    |   movel(pose_trans(ref_frame,p[0.110397, 0.057635, -0.000125, -0.013708, 3.141563, -0.000000]),accel_mss,speed_ms,0,0.001)
    |   movel(pose_trans(ref_frame,p[0.110185, 0.057584, -0.000125, -0.013708, 3.141563, -0.000000]),accel_mss,speed_ms,0,0.001)
    |   movel(pose_trans(ref_frame,p[0.106841, 0.057587, -0.000125, -0.013708, 3.141563, -0.000000]),accel_mss,speed_ms,0,0.001)
    |   movel(pose_trans(ref_frame,p[0.103498, 0.057593, -0.000125, -0.013708, 3.141563, -0.000000]),accel_mss,speed_ms,0,0.001)
    |   movel(pose_trans(ref_frame,p[0.100318, 0.057604, -0.000125, -0.013708, 3.141563, -0.000000]),accel_mss,speed_ms,0,0.001)
    |   movel(pose_trans(ref_frame,p[0.097137, 0.057625, -0.000125, -0.013708, 3.141563, 0.000000]),accel_mss,speed_ms,0,0.001)
    |   movel(pose_trans(ref_frame,p[0.096513, 0.057673, -0.000125, -0.013708, 3.141563, 0.000000]),accel_mss,speed_ms,0,0.001)
    |   movel(pose_trans(ref_frame,p[0.095902, 0.057808, -0.000125, -0.013708, 3.141563, 0.000000]),accel_mss,speed_ms,0,0.001)
    |   movel(pose_trans(ref_frame,p[0.094724, 0.058284, -0.000125, -0.013708, 3.141563, -0.000000]),accel_mss,speed_ms,0,0.001)
    |   movel(pose_trans(ref_frame,p[0.093662, 0.058981, -0.000125, -0.013708, 3.141563, 0.000000]),accel_mss,speed_ms,0,0.001)
    |   movel(pose_trans(ref_frame,p[0.092768, 0.059865, -0.000125, -0.013708, 3.141563, -0.000000]),accel_mss,speed_ms,0,0.001)
    |   movel(pose_trans(ref_frame,p[0.092068, 0.060911, -0.000125, -0.013708, 3.141563, -0.000000]),accel_mss,speed_ms,0,0.001)
    |   movel(pose_trans(ref_frame,p[0.091599, 0.062063, -0.000125, -0.013708, 3.141563, -0.000000]),accel_mss,speed_ms,0,0.001)
    |   movel(pose_trans(ref_frame,p[0.091375, 0.063287, -0.000125, -0.013708, 3.141563, 0.000000]),accel_mss,speed_ms,0,0.001)
    |   movel(pose_trans(ref_frame,p[0.091405, 0.064523, -0.000125, -0.013708, 3.141563, 0.000000]),accel_mss,speed_ms,0,0.001)
    |   movel(pose_trans(ref_frame,p[0.091691, 0.065727, -0.000125, -0.013708, 3.141563, 0.000000]),accel_mss,speed_ms,0,0.001)
    |   movel(pose_trans(ref_frame,p[0.091870, 0.066190, -0.000125, -0.013708, 3.141563, -0.000000]),accel_mss,speed_ms,0,0.001)
    |   movel(pose_trans(ref_frame,p[0.092079, 0.066640, -0.000125, -0.013708, 3.141563, -0.000000]),accel_mss,speed_ms,0,0.001)
    |   movel(pose_trans(ref_frame,p[0.092300, 0.067034, -0.000125, -0.013708, 3.141563, -0.000000]),accel_mss,speed_ms,0,0.001)
    |   movel(pose_trans(ref_frame,p[0.092554, 0.067407, -0.000125, -0.013708, 3.141563, -0.000000]),accel_mss,speed_ms,0,0.001)
    |   movel(pose_trans(ref_frame,p[0.092839, 0.067757, -0.000125, -0.013708, 3.141563, -0.000000]),accel_mss,speed_ms,0,0.001)
    |   movel(pose_trans(ref_frame,p[0.093154, 0.068082, -0.000125, -0.013708, 3.141563, -0.000000]),accel_mss,speed_ms,0,0.001)
    |   movel(pose_trans(ref_frame,p[0.093526, 0.068412, -0.000125, -0.013708, 3.141563, -0.000000]),accel_mss,speed_ms,0,0.001)
    |   movel(pose_trans(ref_frame,p[0.093919, 0.068718, -0.000125, -0.013708, 3.141563, -0.000000]),accel_mss,speed_ms,0,0) # end trace
    |   speed_ms    = 1.000
    |   movel(pose_trans(ref_frame,p[0.093921, 0.068718, 0.005000, -0.013708, 3.141563, -0.000000]),accel_mss,speed_ms,0,0.001)
    |   movel(pose_trans(ref_frame,p[0.109466, 0.038489, 0.005000, -0.013708, 3.141563, -0.000000]),accel_mss,speed_ms,0,0) # end trace
    |   speed_ms    = 0.002
    |   movel(pose_trans(ref_frame,p[0.109466, 0.038489, -0.000125, -0.013708, 3.141563, 0.000000]),accel_mss,speed_ms,0,0) # end trace
    |   speed_ms    = 0.007
    |   movel(pose_trans(ref_frame,p[0.109569, 0.038507, -0.000125, -0.013708, 3.141563, -0.000000]),accel_mss,speed_ms,0,0.001)
    |   movel(pose_trans(ref_frame,p[0.109673, 0.038505, -0.000125, -0.013708, 3.141563, 0.000000]),accel_mss,speed_ms,0,0.001)
    |   movel(pose_trans(ref_frame,p[0.109805, 0.038481, -0.000125, -0.013708, 3.141563, -0.000000]),accel_mss,speed_ms,0,0.001)
    |   movel(pose_trans(ref_frame,p[0.109934, 0.038445, -0.000125, -0.013708, 3.141563, -0.000000]),accel_mss,speed_ms,0,0.001)
    |   movel(pose_trans(ref_frame,p[0.110111, 0.038380, -0.000125, -0.013708, 3.141563, -0.000000]),accel_mss,speed_ms,0,0.001)
    |   movel(pose_trans(ref_frame,p[0.110284, 0.038303, -0.000125, -0.013708, 3.141563, -0.000000]),accel_mss,speed_ms,0,0.001)
    |   movel(pose_trans(ref_frame,p[0.110541, 0.038176, -0.000125, -0.013708, 3.141563, -0.000000]),accel_mss,speed_ms,0,0.001)
    |   movel(pose_trans(ref_frame,p[0.110795, 0.038045, -0.000125, -0.013708, 3.141563, -0.000000]),accel_mss,speed_ms,0,0.001)
    |   movel(pose_trans(ref_frame,p[0.111492, 0.037703, -0.000125, -0.013708, 3.141563, -0.000000]),accel_mss,speed_ms,0,0.001)
    |   movel(pose_trans(ref_frame,p[0.112210, 0.037408, -0.000125, -0.013708, 3.141563, 0.000000]),accel_mss,speed_ms,0,0.001)
    |   movel(pose_trans(ref_frame,p[0.112732, 0.037267, -0.000125, -0.013708, 3.141563, -0.000000]),accel_mss,speed_ms,0,0.001)
    |   movel(pose_trans(ref_frame,p[0.113270, 0.037223, -0.000125, -0.013708, 3.141563, 0.000000]),accel_mss,speed_ms,0,0.001)
    |   movel(pose_trans(ref_frame,p[0.113818, 0.037279, -0.000125, -0.013708, 3.141563, -0.000000]),accel_mss,speed_ms,0,0.001)
    |   movel(pose_trans(ref_frame,p[0.114348, 0.037432, -0.000125, -0.013708, 3.141563, -0.000000]),accel_mss,speed_ms,0,0.001)
    |   movel(pose_trans(ref_frame,p[0.115100, 0.037748, -0.000125, -0.013708, 3.141563, 0.000000]),accel_mss,speed_ms,0,0.001)
    |   movel(pose_trans(ref_frame,p[0.115833, 0.038108, -0.000125, -0.013708, 3.141563, -0.000000]),accel_mss,speed_ms,0,0.001)
    |   movel(pose_trans(ref_frame,p[0.116136, 0.038265, -0.000125, -0.013708, 3.141563, 0.000000]),accel_mss,speed_ms,0,0.001)
    |   movel(pose_trans(ref_frame,p[0.116441, 0.038419, -0.000125, -0.013708, 3.141563, -0.000000]),accel_mss,speed_ms,0,0.001)
    |   movel(pose_trans(ref_frame,p[0.116571, 0.038472, -0.000125, -0.013708, 3.141563, -0.000000]),accel_mss,speed_ms,0,0.001)
    |   movel(pose_trans(ref_frame,p[0.116708, 0.038508, -0.000125, -0.013708, 3.141563, 0.000000]),accel_mss,speed_ms,0,0.001)
    |   movel(pose_trans(ref_frame,p[0.116813, 0.038515, -0.000125, -0.013708, 3.141563, -0.000000]),accel_mss,speed_ms,0,0.001)
    |   movel(pose_trans(ref_frame,p[0.116916, 0.038493, -0.000125, -0.013708, 3.141563, 0.000000]),accel_mss,speed_ms,0,0.001)
    |   movel(pose_trans(ref_frame,p[0.117051, 0.038438, -0.000125, -0.013708, 3.141563, 0.000000]),accel_mss,speed_ms,0,0.001)
    |   movel(pose_trans(ref_frame,p[0.117180, 0.038369, -0.000125, -0.013708, 3.141563, 0.000000]),accel_mss,speed_ms,0,0.001)
    |   movel(pose_trans(ref_frame,p[0.117339, 0.038252, -0.000125, -0.013708, 3.141563, -0.000000]),accel_mss,speed_ms,0,0.001)
    |   movel(pose_trans(ref_frame,p[0.117471, 0.038106, -0.000125, -0.013708, 3.141563, -0.000000]),accel_mss,speed_ms,0,0.001)
    |   movel(pose_trans(ref_frame,p[0.117545, 0.037961, -0.000125, -0.013708, 3.141563, -0.000000]),accel_mss,speed_ms,0,0.001)
    |   movel(pose_trans(ref_frame,p[0.117566, 0.037799, -0.000125, -0.013708, 3.141563, 0.000000]),accel_mss,speed_ms,0,0.001)
    |   movel(pose_trans(ref_frame,p[0.117537, 0.037580, -0.000125, -0.013708, 3.141563, 0.000000]),accel_mss,speed_ms,0,0.001)
    |   movel(pose_trans(ref_frame,p[0.117466, 0.037370, -0.000125, -0.013708, 3.141563, 0.000000]),accel_mss,speed_ms,0,0.001)
    |   movel(pose_trans(ref_frame,p[0.117297, 0.037011, -0.000125, -0.013708, 3.141563, -0.000000]),accel_mss,speed_ms,0,0.001)
    |   movel(pose_trans(ref_frame,p[0.117115, 0.036659, -0.000125, -0.013708, 3.141563, -0.000000]),accel_mss,speed_ms,0,0.001)
    |   movel(pose_trans(ref_frame,p[0.116779, 0.035981, -0.000125, -0.013708, 3.141563, -0.000000]),accel_mss,speed_ms,0,0.001)
    |   movel(pose_trans(ref_frame,p[0.116493, 0.035281, -0.000125, -0.013708, 3.141563, -0.000000]),accel_mss,speed_ms,0,0.001)
    |   movel(pose_trans(ref_frame,p[0.116347, 0.034741, -0.000125, -0.013708, 3.141563, -0.000000]),accel_mss,speed_ms,0,0.001)
    |   movel(pose_trans(ref_frame,p[0.116298, 0.034183, -0.000125, -0.013708, 3.141563, -0.000000]),accel_mss,speed_ms,0,0.001)
    |   movel(pose_trans(ref_frame,p[0.116347, 0.033625, -0.000125, -0.013708, 3.141563, -0.000000]),accel_mss,speed_ms,0,0.001)
    |   movel(pose_trans(ref_frame,p[0.116492, 0.033084, -0.000125, -0.013708, 3.141563, -0.000000]),accel_mss,speed_ms,0,0.001)
    |   movel(pose_trans(ref_frame,p[0.116778, 0.032382, -0.000125, -0.013708, 3.141563, 0.000000]),accel_mss,speed_ms,0,0.001)
    |   movel(pose_trans(ref_frame,p[0.117114, 0.031703, -0.000125, -0.013708, 3.141563, 0.000000]),accel_mss,speed_ms,0,0.001)
    |   movel(pose_trans(ref_frame,p[0.117282, 0.031378, -0.000125, -0.013708, 3.141563, -0.000000]),accel_mss,speed_ms,0,0.001)
    |   movel(pose_trans(ref_frame,p[0.117440, 0.031048, -0.000125, -0.013708, 3.141563, -0.000000]),accel_mss,speed_ms,0,0.001)
    |   movel(pose_trans(ref_frame,p[0.117514, 0.030847, -0.000125, -0.013708, 3.141563, -0.000000]),accel_mss,speed_ms,0,0.001)
    |   movel(pose_trans(ref_frame,p[0.117557, 0.030638, -0.000125, -0.013708, 3.141563, -0.000000]),accel_mss,speed_ms,0,0.001)
    |   movel(pose_trans(ref_frame,p[0.117557, 0.030481, -0.000125, -0.013708, 3.141563, 0.000000]),accel_mss,speed_ms,0,0.001)
    |   movel(pose_trans(ref_frame,p[0.117517, 0.030329, -0.000125, -0.013708, 3.141563, -0.000000]),accel_mss,speed_ms,0,0.001)
    |   movel(pose_trans(ref_frame,p[0.117437, 0.030178, -0.000125, -0.013708, 3.141563, -0.000000]),accel_mss,speed_ms,0,0.001)
    |   movel(pose_trans(ref_frame,p[0.117328, 0.030045, -0.000125, -0.013708, 3.141563, -0.000000]),accel_mss,speed_ms,0,0.001)
    |   movel(pose_trans(ref_frame,p[0.117199, 0.029939, -0.000125, -0.013708, 3.141563, -0.000000]),accel_mss,speed_ms,0,0.001)
    |   movel(pose_trans(ref_frame,p[0.117052, 0.029858, -0.000125, -0.013708, 3.141563, -0.000000]),accel_mss,speed_ms,0,0.001)
    |   movel(pose_trans(ref_frame,p[0.116906, 0.029817, -0.000125, -0.013708, 3.141563, -0.000000]),accel_mss,speed_ms,0,0.001)
    |   movel(pose_trans(ref_frame,p[0.116754, 0.029814, -0.000125, -0.013708, 3.141563, -0.000000]),accel_mss,speed_ms,0,0.001)
    |   movel(pose_trans(ref_frame,p[0.116560, 0.029851, -0.000125, -0.013708, 3.141563, -0.000000]),accel_mss,speed_ms,0,0.001)
    |   movel(pose_trans(ref_frame,p[0.116375, 0.029919, -0.000125, -0.013708, 3.141563, -0.000000]),accel_mss,speed_ms,0,0.001)
    |   movel(pose_trans(ref_frame,p[0.116090, 0.030059, -0.000125, -0.013708, 3.141563, -0.000000]),accel_mss,speed_ms,0,0.001)
    |   movel(pose_trans(ref_frame,p[0.115811, 0.030210, -0.000125, -0.013708, 3.141563, -0.000000]),accel_mss,speed_ms,0,0.001)
    |   movel(pose_trans(ref_frame,p[0.115108, 0.030574, -0.000125, -0.013708, 3.141563, -0.000000]),accel_mss,speed_ms,0,0.001)
    |   movel(pose_trans(ref_frame,p[0.114378, 0.030879, -0.000125, -0.013708, 3.141563, -0.000000]),accel_mss,speed_ms,0,0.001)
    |   movel(pose_trans(ref_frame,p[0.113793, 0.031038, -0.000125, -0.013708, 3.141563, -0.000000]),accel_mss,speed_ms,0,0.001)
    |   movel(pose_trans(ref_frame,p[0.113189, 0.031091, -0.000125, -0.013708, 3.141563, -0.000000]),accel_mss,speed_ms,0,0.001)
    |   movel(pose_trans(ref_frame,p[0.112583, 0.031035, -0.000125, -0.013708, 3.141563, 0.000000]),accel_mss,speed_ms,0,0.001)
    |   movel(pose_trans(ref_frame,p[0.111996, 0.030873, -0.000125, -0.013708, 3.141563, 0.000000]),accel_mss,speed_ms,0,0.001)
    |   movel(pose_trans(ref_frame,p[0.111259, 0.030562, -0.000125, -0.013708, 3.141563, -0.000000]),accel_mss,speed_ms,0,0.001)
    |   movel(pose_trans(ref_frame,p[0.110548, 0.030194, -0.000125, -0.013708, 3.141563, 0.000000]),accel_mss,speed_ms,0,0.001)
    |   movel(pose_trans(ref_frame,p[0.110336, 0.030076, -0.000125, -0.013708, 3.141563, -0.000000]),accel_mss,speed_ms,0,0.001)
    |   movel(pose_trans(ref_frame,p[0.110121, 0.029964, -0.000125, -0.013708, 3.141563, 0.000000]),accel_mss,speed_ms,0,0.001)
    |   movel(pose_trans(ref_frame,p[0.109993, 0.029908, -0.000125, -0.013708, 3.141563, -0.000000]),accel_mss,speed_ms,0,0.001)
    |   movel(pose_trans(ref_frame,p[0.109860, 0.029867, -0.000125, -0.013708, 3.141563, -0.000000]),accel_mss,speed_ms,0,0.001)
    |   movel(pose_trans(ref_frame,p[0.109751, 0.029851, -0.000125, -0.013708, 3.141563, -0.000000]),accel_mss,speed_ms,0,0.001)
    |   movel(pose_trans(ref_frame,p[0.109641, 0.029854, -0.000125, -0.013708, 3.141563, -0.000000]),accel_mss,speed_ms,0,0.001)
    |   movel(pose_trans(ref_frame,p[0.109514, 0.029876, -0.000125, -0.013708, 3.141563, 0.000000]),accel_mss,speed_ms,0,0.001)
    |   movel(pose_trans(ref_frame,p[0.109390, 0.029912, -0.000125, -0.013708, 3.141563, 0.000000]),accel_mss,speed_ms,0,0.001)
    |   movel(pose_trans(ref_frame,p[0.109202, 0.030005, -0.000125, -0.013708, 3.141563, -0.000000]),accel_mss,speed_ms,0,0.001)
    |   movel(pose_trans(ref_frame,p[0.109041, 0.030140, -0.000125, -0.013708, 3.141563, -0.000000]),accel_mss,speed_ms,0,0.001)
    |   movel(pose_trans(ref_frame,p[0.108941, 0.030294, -0.000125, -0.013708, 3.141563, -0.000000]),accel_mss,speed_ms,0,0.001)
    |   movel(pose_trans(ref_frame,p[0.108901, 0.030473, -0.000125, -0.013708, 3.141563, -0.000000]),accel_mss,speed_ms,0,0.001)
    |   movel(pose_trans(ref_frame,p[0.108918, 0.030719, -0.000125, -0.013708, 3.141563, 0.000000]),accel_mss,speed_ms,0,0.001)
    |   movel(pose_trans(ref_frame,p[0.108985, 0.030956, -0.000125, -0.013708, 3.141563, 0.000000]),accel_mss,speed_ms,0,0.001)
    |   movel(pose_trans(ref_frame,p[0.109141, 0.031313, -0.000125, -0.013708, 3.141563, -0.000000]),accel_mss,speed_ms,0,0.001)
    |   movel(pose_trans(ref_frame,p[0.109318, 0.031660, -0.000125, -0.013708, 3.141563, 0.000000]),accel_mss,speed_ms,0,0.001)
    |   movel(pose_trans(ref_frame,p[0.109510, 0.032028, -0.000125, -0.013708, 3.141563, -0.000000]),accel_mss,speed_ms,0,0.001)
    |   movel(pose_trans(ref_frame,p[0.109687, 0.032403, -0.000125, -0.013708, 3.141563, -0.000000]),accel_mss,speed_ms,0,0.001)
    |   movel(pose_trans(ref_frame,p[0.109831, 0.032751, -0.000125, -0.013708, 3.141563, -0.000000]),accel_mss,speed_ms,0,0.001)
    |   movel(pose_trans(ref_frame,p[0.109958, 0.033105, -0.000125, -0.013708, 3.141563, -0.000000]),accel_mss,speed_ms,0,0.001)
    |   movel(pose_trans(ref_frame,p[0.110049, 0.033417, -0.000125, -0.013708, 3.141563, -0.000000]),accel_mss,speed_ms,0,0.001)
    |   movel(pose_trans(ref_frame,p[0.110122, 0.033734, -0.000125, -0.013708, 3.141563, -0.000000]),accel_mss,speed_ms,0,0.001)
    |   movel(pose_trans(ref_frame,p[0.110157, 0.033990, -0.000125, -0.013708, 3.141563, 0.000000]),accel_mss,speed_ms,0,0.001)
    |   movel(pose_trans(ref_frame,p[0.110163, 0.034250, -0.000125, -0.013708, 3.141563, -0.000000]),accel_mss,speed_ms,0,0.001)
    |   movel(pose_trans(ref_frame,p[0.110141, 0.034510, -0.000125, -0.013708, 3.141563, 0.000000]),accel_mss,speed_ms,0,0.001)
    |   movel(pose_trans(ref_frame,p[0.110094, 0.034768, -0.000125, -0.013708, 3.141563, -0.000000]),accel_mss,speed_ms,0,0.001)
    |   movel(pose_trans(ref_frame,p[0.110012, 0.035080, -0.000125, -0.013708, 3.141563, -0.000000]),accel_mss,speed_ms,0,0.001)
    |   movel(pose_trans(ref_frame,p[0.109915, 0.035388, -0.000125, -0.013708, 3.141563, -0.000000]),accel_mss,speed_ms,0,0.001)
    |   movel(pose_trans(ref_frame,p[0.109790, 0.035722, -0.000125, -0.013708, 3.141563, -0.000000]),accel_mss,speed_ms,0,0.001)
    |   movel(pose_trans(ref_frame,p[0.109649, 0.036050, -0.000125, -0.013708, 3.141563, -0.000000]),accel_mss,speed_ms,0,0.001)
    |   movel(pose_trans(ref_frame,p[0.109489, 0.036379, -0.000125, -0.013708, 3.141563, -0.000000]),accel_mss,speed_ms,0,0.001)
    |   movel(pose_trans(ref_frame,p[0.109315, 0.036701, -0.000125, -0.013708, 3.141563, 0.000000]),accel_mss,speed_ms,0,0.001)
    |   movel(pose_trans(ref_frame,p[0.109172, 0.036957, -0.000125, -0.013708, 3.141563, 0.000000]),accel_mss,speed_ms,0,0.001)
    |   movel(pose_trans(ref_frame,p[0.109037, 0.037217, -0.000125, -0.013708, 3.141563, -0.000000]),accel_mss,speed_ms,0,0.001)
    |   movel(pose_trans(ref_frame,p[0.108967, 0.037375, -0.000125, -0.013708, 3.141563, -0.000000]),accel_mss,speed_ms,0,0.001)
    |   movel(pose_trans(ref_frame,p[0.108914, 0.037540, -0.000125, -0.013708, 3.141563, -0.000000]),accel_mss,speed_ms,0,0.001)
    |   movel(pose_trans(ref_frame,p[0.108893, 0.037668, -0.000125, -0.013708, 3.141563, 0.000000]),accel_mss,speed_ms,0,0.001)
    |   movel(pose_trans(ref_frame,p[0.108895, 0.037798, -0.000125, -0.013708, 3.141563, -0.000000]),accel_mss,speed_ms,0,0.001)
    |   movel(pose_trans(ref_frame,p[0.108919, 0.037933, -0.000125, -0.013708, 3.141563, -0.000000]),accel_mss,speed_ms,0,0.001)
    |   movel(pose_trans(ref_frame,p[0.108963, 0.038063, -0.000125, -0.013708, 3.141563, 0.000000]),accel_mss,speed_ms,0,0.001)
    |   movel(pose_trans(ref_frame,p[0.109009, 0.038166, -0.000125, -0.013708, 3.141563, 0.000000]),accel_mss,speed_ms,0,0.001)
    |   movel(pose_trans(ref_frame,p[0.109057, 0.038268, -0.000125, -0.013708, 3.141563, -0.000000]),accel_mss,speed_ms,0,0.001)
    |   movel(pose_trans(ref_frame,p[0.109088, 0.038316, -0.000125, -0.013708, 3.141563, -0.000000]),accel_mss,speed_ms,0,0.001)
    |   movel(pose_trans(ref_frame,p[0.109127, 0.038357, -0.000125, -0.013708, 3.141563, -0.000000]),accel_mss,speed_ms,0,0.001)
    |   movel(pose_trans(ref_frame,p[0.109175, 0.038390, -0.000125, -0.013708, 3.141563, 0.000000]),accel_mss,speed_ms,0,0.001)
    |   movel(pose_trans(ref_frame,p[0.109228, 0.038414, -0.000125, -0.013708, 3.141563, -0.000000]),accel_mss,speed_ms,0,0.001)
    |   movel(pose_trans(ref_frame,p[0.109347, 0.038453, -0.000125, -0.013708, 3.141563, -0.000000]),accel_mss,speed_ms,0,0.001)
    |   movel(pose_trans(ref_frame,p[0.109466, 0.038489, -0.000125, -0.013708, 3.141563, -0.000000]),accel_mss,speed_ms,0,0) # end trace
    |   speed_ms    = 1.000
    |   movel(pose_trans(ref_frame,p[0.109466, 0.038489, 0.005000, -0.013708, 3.141563, -0.000000]),accel_mss,speed_ms,0,0.001)
    |   movel(pose_trans(ref_frame,p[0.035021, 0.042217, 0.005000, -0.013708, 3.141563, -0.000000]),accel_mss,speed_ms,0,0) # end trace
    |   speed_ms    = 0.002
    |   movel(pose_trans(ref_frame,p[0.035021, 0.042217, -0.000125, -0.013708, 3.141563, -0.000000]),accel_mss,speed_ms,0,0) # end trace
    |   speed_ms    = 0.007
    |   movel(pose_trans(ref_frame,p[0.035696, 0.042643, -0.000125, -0.013708, 3.141563, -0.000000]),accel_mss,speed_ms,0,0.001)
    |   movel(pose_trans(ref_frame,p[0.036424, 0.042969, -0.000125, -0.013708, 3.141563, 0.000000]),accel_mss,speed_ms,0,0.001)
    |   movel(pose_trans(ref_frame,p[0.037174, 0.043179, -0.000125, -0.013708, 3.141563, -0.000000]),accel_mss,speed_ms,0,0.001)
    |   movel(pose_trans(ref_frame,p[0.037947, 0.043271, -0.000125, -0.013708, 3.141563, 0.000000]),accel_mss,speed_ms,0,0.001)
    |   movel(pose_trans(ref_frame,p[0.038764, 0.043248, -0.000125, -0.013708, 3.141563, -0.000000]),accel_mss,speed_ms,0,0.001)
    |   movel(pose_trans(ref_frame,p[0.039570, 0.043107, -0.000125, -0.013708, 3.141563, 0.000000]),accel_mss,speed_ms,0,0.001)
    |   movel(pose_trans(ref_frame,p[0.040436, 0.042841, -0.000125, -0.013708, 3.141563, -0.000000]),accel_mss,speed_ms,0,0.001)
    |   movel(pose_trans(ref_frame,p[0.041269, 0.042485, -0.000125, -0.013708, 3.141563, -0.000000]),accel_mss,speed_ms,0,0.001)
    |   movel(pose_trans(ref_frame,p[0.041570, 0.042331, -0.000125, -0.013708, 3.141563, 0.000000]),accel_mss,speed_ms,0,0.001)
    |   movel(pose_trans(ref_frame,p[0.041866, 0.042166, -0.000125, -0.013708, 3.141563, 0.000000]),accel_mss,speed_ms,0,0.001)
    |   movel(pose_trans(ref_frame,p[0.042087, 0.042027, -0.000125, -0.013708, 3.141563, -0.000000]),accel_mss,speed_ms,0,0.001)
    |   movel(pose_trans(ref_frame,p[0.042298, 0.041872, -0.000125, -0.013708, 3.141563, -0.000000]),accel_mss,speed_ms,0,0.001)
    |   movel(pose_trans(ref_frame,p[0.042544, 0.041666, -0.000125, -0.013708, 3.141563, 0.000000]),accel_mss,speed_ms,0,0.001)
    |   movel(pose_trans(ref_frame,p[0.042782, 0.041448, -0.000125, -0.013708, 3.141563, 0.000000]),accel_mss,speed_ms,0,0.001)
    |   movel(pose_trans(ref_frame,p[0.043232, 0.041011, -0.000125, -0.013708, 3.141563, 0.000000]),accel_mss,speed_ms,0,0.001)
    |   movel(pose_trans(ref_frame,p[0.043678, 0.040571, -0.000125, -0.013708, 3.141563, -0.000000]),accel_mss,speed_ms,0,0.001)
    |   movel(pose_trans(ref_frame,p[0.044126, 0.040122, -0.000125, -0.013708, 3.141563, -0.000000]),accel_mss,speed_ms,0,0.001)
    |   movel(pose_trans(ref_frame,p[0.044571, 0.039671, -0.000125, -0.013708, 3.141563, -0.000000]),accel_mss,speed_ms,0,0.001)
    |   movel(pose_trans(ref_frame,p[0.044790, 0.039435, -0.000125, -0.013708, 3.141563, -0.000000]),accel_mss,speed_ms,0,0.001)
    |   movel(pose_trans(ref_frame,p[0.044998, 0.039188, -0.000125, -0.013708, 3.141563, 0.000000]),accel_mss,speed_ms,0,0.001)
    |   movel(pose_trans(ref_frame,p[0.045157, 0.038974, -0.000125, -0.013708, 3.141563, -0.000000]),accel_mss,speed_ms,0,0.001)
    |   movel(pose_trans(ref_frame,p[0.045300, 0.038749, -0.000125, -0.013708, 3.141563, -0.000000]),accel_mss,speed_ms,0,0.001)
    |   movel(pose_trans(ref_frame,p[0.045478, 0.038435, -0.000125, -0.013708, 3.141563, 0.000000]),accel_mss,speed_ms,0,0.001)
    |   movel(pose_trans(ref_frame,p[0.045646, 0.038116, -0.000125, -0.013708, 3.141563, 0.000000]),accel_mss,speed_ms,0,0.001)
    |   movel(pose_trans(ref_frame,p[0.046037, 0.037220, -0.000125, -0.013708, 3.141563, -0.000000]),accel_mss,speed_ms,0,0.001)
    |   movel(pose_trans(ref_frame,p[0.046320, 0.036284, -0.000125, -0.013708, 3.141563, -0.000000]),accel_mss,speed_ms,0,0.001)
    |   movel(pose_trans(ref_frame,p[0.046458, 0.035405, -0.000125, -0.013708, 3.141563, -0.000000]),accel_mss,speed_ms,0,0.001)
    |   movel(pose_trans(ref_frame,p[0.046457, 0.034516, -0.000125, -0.013708, 3.141563, -0.000000]),accel_mss,speed_ms,0,0.001)
    |   movel(pose_trans(ref_frame,p[0.046319, 0.033675, -0.000125, -0.013708, 3.141563, -0.000000]),accel_mss,speed_ms,0,0.001)
    |   movel(pose_trans(ref_frame,p[0.046045, 0.032869, -0.000125, -0.013708, 3.141563, 0.000000]),accel_mss,speed_ms,0,0.001)
    |   movel(pose_trans(ref_frame,p[0.045635, 0.032095, -0.000125, -0.013708, 3.141563, 0.000000]),accel_mss,speed_ms,0,0.001)
    |   movel(pose_trans(ref_frame,p[0.045112, 0.031391, -0.000125, -0.013708, 3.141563, -0.000000]),accel_mss,speed_ms,0,0.001)
    |   movel(pose_trans(ref_frame,p[0.044169, 0.030532, -0.000125, -0.013708, 3.141563, -0.000000]),accel_mss,speed_ms,0,0.001)
    |   movel(pose_trans(ref_frame,p[0.043053, 0.029913, -0.000125, -0.013708, 3.141563, -0.000000]),accel_mss,speed_ms,0,0.001)
    |   movel(pose_trans(ref_frame,p[0.041835, 0.029576, -0.000125, -0.013708, 3.141563, -0.000000]),accel_mss,speed_ms,0,0.001)
    |   movel(pose_trans(ref_frame,p[0.040572, 0.029537, -0.000125, -0.013708, 3.141563, 0.000000]),accel_mss,speed_ms,0,0.001)
    |   movel(pose_trans(ref_frame,p[0.039201, 0.029806, -0.000125, -0.013708, 3.141563, 0.000000]),accel_mss,speed_ms,0,0.001)
    |   movel(pose_trans(ref_frame,p[0.037915, 0.030351, -0.000125, -0.013708, 3.141563, 0.000000]),accel_mss,speed_ms,0,0.001)
    |   movel(pose_trans(ref_frame,p[0.036576, 0.031218, -0.000125, -0.013708, 3.141563, -0.000000]),accel_mss,speed_ms,0,0.001)
    |   movel(pose_trans(ref_frame,p[0.035372, 0.032264, -0.000125, -0.013708, 3.141563, 0.000000]),accel_mss,speed_ms,0,0.001)
    |   movel(pose_trans(ref_frame,p[0.034473, 0.033280, -0.000125, -0.013708, 3.141563, 0.000000]),accel_mss,speed_ms,0,0.001)
    |   movel(pose_trans(ref_frame,p[0.033705, 0.034398, -0.000125, -0.013708, 3.141563, 0.000000]),accel_mss,speed_ms,0,0.001)
    |   movel(pose_trans(ref_frame,p[0.033173, 0.035486, -0.000125, -0.013708, 3.141563, -0.000000]),accel_mss,speed_ms,0,0.001)
    |   movel(pose_trans(ref_frame,p[0.032833, 0.036648, -0.000125, -0.013708, 3.141563, 0.000000]),accel_mss,speed_ms,0,0.001)
    |   movel(pose_trans(ref_frame,p[0.032721, 0.037742, -0.000125, -0.013708, 3.141563, 0.000000]),accel_mss,speed_ms,0,0.001)
    |   movel(pose_trans(ref_frame,p[0.032823, 0.038837, -0.000125, -0.013708, 3.141563, 0.000000]),accel_mss,speed_ms,0,0.001)
    |   movel(pose_trans(ref_frame,p[0.033134, 0.039863, -0.000125, -0.013708, 3.141563, -0.000000]),accel_mss,speed_ms,0,0.001)
    |   movel(pose_trans(ref_frame,p[0.033652, 0.040802, -0.000125, -0.013708, 3.141563, 0.000000]),accel_mss,speed_ms,0,0.001)
    |   movel(pose_trans(ref_frame,p[0.033848, 0.041082, -0.000125, -0.013708, 3.141563, 0.000000]),accel_mss,speed_ms,0,0.001)
    |   movel(pose_trans(ref_frame,p[0.034047, 0.041359, -0.000125, -0.013708, 3.141563, 0.000000]),accel_mss,speed_ms,0,0.001)
    |   movel(pose_trans(ref_frame,p[0.034147, 0.041487, -0.000125, -0.013708, 3.141563, -0.000000]),accel_mss,speed_ms,0,0.001)
    |   movel(pose_trans(ref_frame,p[0.034256, 0.041608, -0.000125, -0.013708, 3.141563, 0.000000]),accel_mss,speed_ms,0,0.001)
    |   movel(pose_trans(ref_frame,p[0.034372, 0.041719, -0.000125, -0.013708, 3.141563, 0.000000]),accel_mss,speed_ms,0,0.001)
    |   movel(pose_trans(ref_frame,p[0.034496, 0.041821, -0.000125, -0.013708, 3.141563, -0.000000]),accel_mss,speed_ms,0,0.001)
    |   movel(pose_trans(ref_frame,p[0.034757, 0.042020, -0.000125, -0.013708, 3.141563, -0.000000]),accel_mss,speed_ms,0,0.001)
    |   movel(pose_trans(ref_frame,p[0.035021, 0.042217, -0.000125, -0.013708, 3.141563, -0.000000]),accel_mss,speed_ms,0,0) # end trace
    |   speed_ms    = 1.000
    |   movel(pose_trans(ref_frame,p[0.035021, 0.042217, 0.005000, -0.013708, 3.141563, -0.000000]),accel_mss,speed_ms,0,0.001)
    |   movel(pose_trans(ref_frame,p[0.034887, 0.040550, 0.005000, -0.013708, 3.141563, 0.000000]),accel_mss,speed_ms,0,0) # end trace
    |   speed_ms    = 0.002
    |   movel(pose_trans(ref_frame,p[0.034887, 0.040550, -0.000125, -0.013708, 3.141563, 0.000000]),accel_mss,speed_ms,0,0) # end trace
    |   speed_ms    = 0.007
    |   movel(pose_trans(ref_frame,p[0.034858, 0.040183, -0.000125, -0.013708, 3.141563, 0.000000]),accel_mss,speed_ms,0,0.001)
    |   movel(pose_trans(ref_frame,p[0.034959, 0.039829, -0.000125, -0.013708, 3.141563, 0.000000]),accel_mss,speed_ms,0,0.001)
    |   movel(pose_trans(ref_frame,p[0.035252, 0.039292, -0.000125, -0.013708, 3.141563, 0.000000]),accel_mss,speed_ms,0,0.001)
    |   movel(pose_trans(ref_frame,p[0.035590, 0.038782, -0.000125, -0.013708, 3.141563, 0.000000]),accel_mss,speed_ms,0,0.001)
    |   movel(pose_trans(ref_frame,p[0.036143, 0.038068, -0.000125, -0.013708, 3.141563, 0.000000]),accel_mss,speed_ms,0,0.001)
    |   movel(pose_trans(ref_frame,p[0.036737, 0.037388, -0.000125, -0.013708, 3.141563, 0.000000]),accel_mss,speed_ms,0,0.001)
    |   movel(pose_trans(ref_frame,p[0.037650, 0.036422, -0.000125, -0.013708, 3.141563, -0.000000]),accel_mss,speed_ms,0,0.001)
    |   movel(pose_trans(ref_frame,p[0.038581, 0.035473, -0.000125, -0.013708, 3.141563, -0.000000]),accel_mss,speed_ms,0,0.001)
    |   movel(pose_trans(ref_frame,p[0.039511, 0.034560, -0.000125, -0.013708, 3.141563, -0.000000]),accel_mss,speed_ms,0,0.001)
    |   movel(pose_trans(ref_frame,p[0.040455, 0.033661, -0.000125, -0.013708, 3.141563, -0.000000]),accel_mss,speed_ms,0,0.001)
    |   movel(pose_trans(ref_frame,p[0.041103, 0.033084, -0.000125, -0.013708, 3.141563, -0.000000]),accel_mss,speed_ms,0,0.001)
    |   movel(pose_trans(ref_frame,p[0.041779, 0.032540, -0.000125, -0.013708, 3.141563, 0.000000]),accel_mss,speed_ms,0,0.001)
    |   movel(pose_trans(ref_frame,p[0.042266, 0.032198, -0.000125, -0.013708, 3.141563, -0.000000]),accel_mss,speed_ms,0,0.001)
    |   movel(pose_trans(ref_frame,p[0.042777, 0.031893, -0.000125, -0.013708, 3.141563, -0.000000]),accel_mss,speed_ms,0,0.001)
    |   movel(pose_trans(ref_frame,p[0.043141, 0.031749, -0.000125, -0.013708, 3.141563, 0.000000]),accel_mss,speed_ms,0,0.001)
    |   movel(pose_trans(ref_frame,p[0.043529, 0.031701, -0.000125, -0.013708, 3.141563, -0.000000]),accel_mss,speed_ms,0,0.001)
    |   movel(pose_trans(ref_frame,p[0.043699, 0.031713, -0.000125, -0.013708, 3.141563, 0.000000]),accel_mss,speed_ms,0,0.001)
    |   movel(pose_trans(ref_frame,p[0.043865, 0.031748, -0.000125, -0.013708, 3.141563, -0.000000]),accel_mss,speed_ms,0,0.001)
    |   movel(pose_trans(ref_frame,p[0.043993, 0.031803, -0.000125, -0.013708, 3.141563, -0.000000]),accel_mss,speed_ms,0,0.001)
    |   movel(pose_trans(ref_frame,p[0.044103, 0.031889, -0.000125, -0.013708, 3.141563, -0.000000]),accel_mss,speed_ms,0,0.001)
    |   movel(pose_trans(ref_frame,p[0.044188, 0.031999, -0.000125, -0.013708, 3.141563, -0.000000]),accel_mss,speed_ms,0,0.001)
    |   movel(pose_trans(ref_frame,p[0.044243, 0.032127, -0.000125, -0.013708, 3.141563, -0.000000]),accel_mss,speed_ms,0,0.001)
    |   movel(pose_trans(ref_frame,p[0.044279, 0.032294, -0.000125, -0.013708, 3.141563, 0.000000]),accel_mss,speed_ms,0,0.001)
    |   movel(pose_trans(ref_frame,p[0.044290, 0.032463, -0.000125, -0.013708, 3.141563, 0.000000]),accel_mss,speed_ms,0,0.001)
    |   movel(pose_trans(ref_frame,p[0.044263, 0.032736, -0.000125, -0.013708, 3.141563, -0.000000]),accel_mss,speed_ms,0,0.001)
    |   movel(pose_trans(ref_frame,p[0.044181, 0.032998, -0.000125, -0.013708, 3.141563, 0.000000]),accel_mss,speed_ms,0,0.001)
    |   movel(pose_trans(ref_frame,p[0.044021, 0.033329, -0.000125, -0.013708, 3.141563, 0.000000]),accel_mss,speed_ms,0,0.001)
    |   movel(pose_trans(ref_frame,p[0.043834, 0.033645, -0.000125, -0.013708, 3.141563, 0.000000]),accel_mss,speed_ms,0,0.001)
    |   movel(pose_trans(ref_frame,p[0.043533, 0.034080, -0.000125, -0.013708, 3.141563, -0.000000]),accel_mss,speed_ms,0,0.001)
    |   movel(pose_trans(ref_frame,p[0.043209, 0.034497, -0.000125, -0.013708, 3.141563, -0.000000]),accel_mss,speed_ms,0,0.001)
    |   movel(pose_trans(ref_frame,p[0.042689, 0.035118, -0.000125, -0.013708, 3.141563, -0.000000]),accel_mss,speed_ms,0,0.001)
    |   movel(pose_trans(ref_frame,p[0.042159, 0.035731, -0.000125, -0.013708, 3.141563, 0.000000]),accel_mss,speed_ms,0,0.001)
    |   movel(pose_trans(ref_frame,p[0.041471, 0.036489, -0.000125, -0.013708, 3.141563, -0.000000]),accel_mss,speed_ms,0,0.001)
    |   movel(pose_trans(ref_frame,p[0.040761, 0.037225, -0.000125, -0.013708, 3.141563, -0.000000]),accel_mss,speed_ms,0,0.001)
    |   movel(pose_trans(ref_frame,p[0.039957, 0.038014, -0.000125, -0.013708, 3.141563, -0.000000]),accel_mss,speed_ms,0,0.001)
    |   movel(pose_trans(ref_frame,p[0.039136, 0.038783, -0.000125, -0.013708, 3.141563, 0.000000]),accel_mss,speed_ms,0,0.001)
    |   movel(pose_trans(ref_frame,p[0.038375, 0.039465, -0.000125, -0.013708, 3.141563, -0.000000]),accel_mss,speed_ms,0,0.001)
    |   movel(pose_trans(ref_frame,p[0.037600, 0.040130, -0.000125, -0.013708, 3.141563, 0.000000]),accel_mss,speed_ms,0,0.001)
    |   movel(pose_trans(ref_frame,p[0.037133, 0.040484, -0.000125, -0.013708, 3.141563, -0.000000]),accel_mss,speed_ms,0,0.001)
    |   movel(pose_trans(ref_frame,p[0.036632, 0.040788, -0.000125, -0.013708, 3.141563, -0.000000]),accel_mss,speed_ms,0,0.001)
    |   movel(pose_trans(ref_frame,p[0.036327, 0.040934, -0.000125, -0.013708, 3.141563, 0.000000]),accel_mss,speed_ms,0,0.001)
    |   movel(pose_trans(ref_frame,p[0.036009, 0.041047, -0.000125, -0.013708, 3.141563, 0.000000]),accel_mss,speed_ms,0,0.001)
    |   movel(pose_trans(ref_frame,p[0.035750, 0.041095, -0.000125, -0.013708, 3.141563, -0.000000]),accel_mss,speed_ms,0,0.001)
    |   movel(pose_trans(ref_frame,p[0.035486, 0.041087, -0.000125, -0.013708, 3.141563, -0.000000]),accel_mss,speed_ms,0,0.001)
    |   movel(pose_trans(ref_frame,p[0.035283, 0.041028, -0.000125, -0.013708, 3.141563, 0.000000]),accel_mss,speed_ms,0,0.001)
    |   movel(pose_trans(ref_frame,p[0.035107, 0.040911, -0.000125, -0.013708, 3.141563, -0.000000]),accel_mss,speed_ms,0,0.001)
    |   movel(pose_trans(ref_frame,p[0.034971, 0.040746, -0.000125, -0.013708, 3.141563, 0.000000]),accel_mss,speed_ms,0,0.001)
    |   movel(pose_trans(ref_frame,p[0.034887, 0.040550, -0.000125, -0.013708, 3.141563, 0.000000]),accel_mss,speed_ms,0,0) # end trace
    |   speed_ms    = 1.000
    |   movel(pose_trans(ref_frame,p[0.034887, 0.040550, 0.005000, -0.013708, 3.141563, 0.000000]),accel_mss,speed_ms,0,0.001)
    |   movel(pose_trans(ref_frame,p[0.026610, 0.033644, 0.005000, -0.013708, 3.141563, -0.000000]),accel_mss,speed_ms,0,0) # end trace
    |   speed_ms    = 0.002
    |   movel(pose_trans(ref_frame,p[0.026610, 0.033644, -0.000125, -0.013708, 3.141563, 0.000000]),accel_mss,speed_ms,0,0) # end trace
    |   speed_ms    = 0.007
    |   movel(pose_trans(ref_frame,p[0.026883, 0.033825, -0.000125, -0.013708, 3.141563, 0.000000]),accel_mss,speed_ms,0,0.001)
    |   movel(pose_trans(ref_frame,p[0.027167, 0.033986, -0.000125, -0.013708, 3.141563, 0.000000]),accel_mss,speed_ms,0,0.001)
    |   movel(pose_trans(ref_frame,p[0.027534, 0.034171, -0.000125, -0.013708, 3.141563, -0.000000]),accel_mss,speed_ms,0,0.001)
    |   movel(pose_trans(ref_frame,p[0.027906, 0.034342, -0.000125, -0.013708, 3.141563, 0.000000]),accel_mss,speed_ms,0,0.001)
    |   movel(pose_trans(ref_frame,p[0.028282, 0.034500, -0.000125, -0.013708, 3.141563, 0.000000]),accel_mss,speed_ms,0,0.001)
    |   movel(pose_trans(ref_frame,p[0.028662, 0.034645, -0.000125, -0.013708, 3.141563, 0.000000]),accel_mss,speed_ms,0,0.001)
    |   movel(pose_trans(ref_frame,p[0.028964, 0.034742, -0.000125, -0.013708, 3.141563, 0.000000]),accel_mss,speed_ms,0,0.001)
    |   movel(pose_trans(ref_frame,p[0.029272, 0.034817, -0.000125, -0.013708, 3.141563, -0.000000]),accel_mss,speed_ms,0,0.001)
    |   movel(pose_trans(ref_frame,p[0.029982, 0.034879, -0.000125, -0.013708, 3.141563, -0.000000]),accel_mss,speed_ms,0,0.001)
    |   movel(pose_trans(ref_frame,p[0.030687, 0.034779, -0.000125, -0.013708, 3.141563, 0.000000]),accel_mss,speed_ms,0,0.001)
    |   movel(pose_trans(ref_frame,p[0.031393, 0.034519, -0.000125, -0.013708, 3.141563, -0.000000]),accel_mss,speed_ms,0,0.001)
    |   movel(pose_trans(ref_frame,p[0.032034, 0.034127, -0.000125, -0.013708, 3.141563, -0.000000]),accel_mss,speed_ms,0,0.001)
    |   movel(pose_trans(ref_frame,p[0.032637, 0.033583, -0.000125, -0.013708, 3.141563, 0.000000]),accel_mss,speed_ms,0,0.001)
    |   movel(pose_trans(ref_frame,p[0.033135, 0.032941, -0.000125, -0.013708, 3.141563, 0.000000]),accel_mss,speed_ms,0,0.001)
    |   movel(pose_trans(ref_frame,p[0.033544, 0.032184, -0.000125, -0.013708, 3.141563, 0.000000]),accel_mss,speed_ms,0,0.001)
    |   movel(pose_trans(ref_frame,p[0.033836, 0.031376, -0.000125, -0.013708, 3.141563, 0.000000]),accel_mss,speed_ms,0,0.001)
    |   movel(pose_trans(ref_frame,p[0.033891, 0.031139, -0.000125, -0.013708, 3.141563, 0.000000]),accel_mss,speed_ms,0,0.001)
    |   movel(pose_trans(ref_frame,p[0.033928, 0.030899, -0.000125, -0.013708, 3.141563, 0.000000]),accel_mss,speed_ms,0,0.001)
    |   movel(pose_trans(ref_frame,p[0.033971, 0.030484, -0.000125, -0.013708, 3.141563, -0.000000]),accel_mss,speed_ms,0,0.001)
    |   movel(pose_trans(ref_frame,p[0.034006, 0.030068, -0.000125, -0.013708, 3.141563, 0.000000]),accel_mss,speed_ms,0,0.001)
    |   movel(pose_trans(ref_frame,p[0.034041, 0.029554, -0.000125, -0.013708, 3.141563, 0.000000]),accel_mss,speed_ms,0,0.001)
    |   movel(pose_trans(ref_frame,p[0.034067, 0.029039, -0.000125, -0.013708, 3.141563, 0.000000]),accel_mss,speed_ms,0,0.001)
    |   movel(pose_trans(ref_frame,p[0.034088, 0.028454, -0.000125, -0.013708, 3.141563, 0.000000]),accel_mss,speed_ms,0,0.001)
    |   movel(pose_trans(ref_frame,p[0.034103, 0.027869, -0.000125, -0.013708, 3.141563, -0.000000]),accel_mss,speed_ms,0,0.001)
    |   movel(pose_trans(ref_frame,p[0.034129, 0.026956, -0.000125, -0.013708, 3.141563, -0.000000]),accel_mss,speed_ms,0,0.001)
    |   movel(pose_trans(ref_frame,p[0.034173, 0.026045, -0.000125, -0.013708, 3.141563, 0.000000]),accel_mss,speed_ms,0,0.001)
    |   movel(pose_trans(ref_frame,p[0.034228, 0.025412, -0.000125, -0.013708, 3.141563, -0.000000]),accel_mss,speed_ms,0,0.001)
    |   movel(pose_trans(ref_frame,p[0.034318, 0.024783, -0.000125, -0.013708, 3.141563, -0.000000]),accel_mss,speed_ms,0,0.001)
    |   movel(pose_trans(ref_frame,p[0.034412, 0.024342, -0.000125, -0.013708, 3.141563, -0.000000]),accel_mss,speed_ms,0,0.001)
    |   movel(pose_trans(ref_frame,p[0.034541, 0.023910, -0.000125, -0.013708, 3.141563, 0.000000]),accel_mss,speed_ms,0,0.001)
    |   movel(pose_trans(ref_frame,p[0.034676, 0.023626, -0.000125, -0.013708, 3.141563, -0.000000]),accel_mss,speed_ms,0,0.001)
    |   movel(pose_trans(ref_frame,p[0.034873, 0.023380, -0.000125, -0.013708, 3.141563, -0.000000]),accel_mss,speed_ms,0,0.001)
    |   movel(pose_trans(ref_frame,p[0.034931, 0.023328, -0.000125, -0.013708, 3.141563, -0.000000]),accel_mss,speed_ms,0,0.001)
    |   movel(pose_trans(ref_frame,p[0.034996, 0.023285, -0.000125, -0.013708, 3.141563, -0.000000]),accel_mss,speed_ms,0,0.001)
    |   movel(pose_trans(ref_frame,p[0.035046, 0.023269, -0.000125, -0.013708, 3.141563, 0.000000]),accel_mss,speed_ms,0,0.001)
    |   movel(pose_trans(ref_frame,p[0.035099, 0.023273, -0.000125, -0.013708, 3.141563, -0.000000]),accel_mss,speed_ms,0,0.001)
    |   movel(pose_trans(ref_frame,p[0.035162, 0.023300, -0.000125, -0.013708, 3.141563, 0.000000]),accel_mss,speed_ms,0,0.001)
    |   movel(pose_trans(ref_frame,p[0.035219, 0.023340, -0.000125, -0.013708, 3.141563, 0.000000]),accel_mss,speed_ms,0,0.001)
    |   movel(pose_trans(ref_frame,p[0.035327, 0.023440, -0.000125, -0.013708, 3.141563, -0.000000]),accel_mss,speed_ms,0,0.001)
    |   movel(pose_trans(ref_frame,p[0.035433, 0.023544, -0.000125, -0.013708, 3.141563, 0.000000]),accel_mss,speed_ms,0,0.001)
    |   movel(pose_trans(ref_frame,p[0.035649, 0.023778, -0.000125, -0.013708, 3.141563, -0.000000]),accel_mss,speed_ms,0,0.001)
    |   movel(pose_trans(ref_frame,p[0.035848, 0.024028, -0.000125, -0.013708, 3.141563, -0.000000]),accel_mss,speed_ms,0,0.001)
    |   movel(pose_trans(ref_frame,p[0.036070, 0.024342, -0.000125, -0.013708, 3.141563, -0.000000]),accel_mss,speed_ms,0,0.001)
    |   movel(pose_trans(ref_frame,p[0.036279, 0.024666, -0.000125, -0.013708, 3.141563, -0.000000]),accel_mss,speed_ms,0,0.001)
    |   movel(pose_trans(ref_frame,p[0.036473, 0.024996, -0.000125, -0.013708, 3.141563, 0.000000]),accel_mss,speed_ms,0,0.001)
    |   movel(pose_trans(ref_frame,p[0.036653, 0.025334, -0.000125, -0.013708, 3.141563, 0.000000]),accel_mss,speed_ms,0,0.001)
    |   movel(pose_trans(ref_frame,p[0.036783, 0.025617, -0.000125, -0.013708, 3.141563, -0.000000]),accel_mss,speed_ms,0,0.001)
    |   movel(pose_trans(ref_frame,p[0.036892, 0.025910, -0.000125, -0.013708, 3.141563, -0.000000]),accel_mss,speed_ms,0,0.001)
    |   movel(pose_trans(ref_frame,p[0.036979, 0.026229, -0.000125, -0.013708, 3.141563, -0.000000]),accel_mss,speed_ms,0,0.001)
    |   movel(pose_trans(ref_frame,p[0.037033, 0.026555, -0.000125, -0.013708, 3.141563, 0.000000]),accel_mss,speed_ms,0,0.001)
    |   movel(pose_trans(ref_frame,p[0.037060, 0.026911, -0.000125, -0.013708, 3.141563, -0.000000]),accel_mss,speed_ms,0,0.001)
    |   movel(pose_trans(ref_frame,p[0.037059, 0.027267, -0.000125, -0.013708, 3.141563, -0.000000]),accel_mss,speed_ms,0,0.001)
    |   movel(pose_trans(ref_frame,p[0.037029, 0.027617, -0.000125, -0.013708, 3.141563, -0.000000]),accel_mss,speed_ms,0,0.001)
    |   movel(pose_trans(ref_frame,p[0.036971, 0.027963, -0.000125, -0.013708, 3.141563, 0.000000]),accel_mss,speed_ms,0,0.001)
    |   movel(pose_trans(ref_frame,p[0.036889, 0.028266, -0.000125, -0.013708, 3.141563, -0.000000]),accel_mss,speed_ms,0,0.001)
    |   movel(pose_trans(ref_frame,p[0.036773, 0.028558, -0.000125, -0.013708, 3.141563, -0.000000]),accel_mss,speed_ms,0,0.001)
    |   movel(pose_trans(ref_frame,p[0.036676, 0.028784, -0.000125, -0.013708, 3.141563, -0.000000]),accel_mss,speed_ms,0,0.001)
    |   movel(pose_trans(ref_frame,p[0.036590, 0.029014, -0.000125, -0.013708, 3.141563, -0.000000]),accel_mss,speed_ms,0,0.001)
    |   movel(pose_trans(ref_frame,p[0.036549, 0.029172, -0.000125, -0.013708, 3.141563, -0.000000]),accel_mss,speed_ms,0,0.001)
    |   movel(pose_trans(ref_frame,p[0.036534, 0.029334, -0.000125, -0.013708, 3.141563, -0.000000]),accel_mss,speed_ms,0,0.001)
    |   movel(pose_trans(ref_frame,p[0.036550, 0.029438, -0.000125, -0.013708, 3.141563, -0.000000]),accel_mss,speed_ms,0,0.001)
    |   movel(pose_trans(ref_frame,p[0.036598, 0.029530, -0.000125, -0.013708, 3.141563, -0.000000]),accel_mss,speed_ms,0,0.001)
    |   movel(pose_trans(ref_frame,p[0.036670, 0.029593, -0.000125, -0.013708, 3.141563, 0.000000]),accel_mss,speed_ms,0,0.001)
    |   movel(pose_trans(ref_frame,p[0.036761, 0.029621, -0.000125, -0.013708, 3.141563, 0.000000]),accel_mss,speed_ms,0,0.001)
    |   movel(pose_trans(ref_frame,p[0.036936, 0.029600, -0.000125, -0.013708, 3.141563, -0.000000]),accel_mss,speed_ms,0,0.001)
    |   movel(pose_trans(ref_frame,p[0.037086, 0.029508, -0.000125, -0.013708, 3.141563, -0.000000]),accel_mss,speed_ms,0,0.001)
    |   movel(pose_trans(ref_frame,p[0.037742, 0.028872, -0.000125, -0.013708, 3.141563, -0.000000]),accel_mss,speed_ms,0,0.001)
    |   movel(pose_trans(ref_frame,p[0.038393, 0.028231, -0.000125, -0.013708, 3.141563, -0.000000]),accel_mss,speed_ms,0,0.001)
    |   movel(pose_trans(ref_frame,p[0.039036, 0.027587, -0.000125, -0.013708, 3.141563, -0.000000]),accel_mss,speed_ms,0,0.001)
    |   movel(pose_trans(ref_frame,p[0.039673, 0.026938, -0.000125, -0.013708, 3.141563, 0.000000]),accel_mss,speed_ms,0,0.001)
    |   movel(pose_trans(ref_frame,p[0.039777, 0.026779, -0.000125, -0.013708, 3.141563, -0.000000]),accel_mss,speed_ms,0,0.001)
    |   movel(pose_trans(ref_frame,p[0.039814, 0.026591, -0.000125, -0.013708, 3.141563, -0.000000]),accel_mss,speed_ms,0,0.001)
    |   movel(pose_trans(ref_frame,p[0.039781, 0.026426, -0.000125, -0.013708, 3.141563, -0.000000]),accel_mss,speed_ms,0,0.001)
    |   movel(pose_trans(ref_frame,p[0.039688, 0.026285, -0.000125, -0.013708, 3.141563, -0.000000]),accel_mss,speed_ms,0,0.001)
    |   movel(pose_trans(ref_frame,p[0.037713, 0.024294, -0.000125, -0.013708, 3.141563, -0.000000]),accel_mss,speed_ms,0,0.001)
    |   movel(pose_trans(ref_frame,p[0.035736, 0.022305, -0.000125, -0.013708, 3.141563, 0.000000]),accel_mss,speed_ms,0,0.001)
    |   movel(pose_trans(ref_frame,p[0.033775, 0.020334, -0.000125, -0.013708, 3.141563, -0.000000]),accel_mss,speed_ms,0,0.001)
    |   movel(pose_trans(ref_frame,p[0.031812, 0.018365, -0.000125, -0.013708, 3.141563, -0.000000]),accel_mss,speed_ms,0,0.001)
    |   movel(pose_trans(ref_frame,p[0.031632, 0.018230, -0.000125, -0.013708, 3.141563, -0.000000]),accel_mss,speed_ms,0,0.001)
    |   movel(pose_trans(ref_frame,p[0.031421, 0.018150, -0.000125, -0.013708, 3.141563, -0.000000]),accel_mss,speed_ms,0,0.001)
    |   movel(pose_trans(ref_frame,p[0.031360, 0.018146, -0.000125, -0.013708, 3.141563, -0.000000]),accel_mss,speed_ms,0,0.001)
    |   movel(pose_trans(ref_frame,p[0.031301, 0.018161, -0.000125, -0.013708, 3.141563, -0.000000]),accel_mss,speed_ms,0,0.001)
    |   movel(pose_trans(ref_frame,p[0.031228, 0.018198, -0.000125, -0.013708, 3.141563, -0.000000]),accel_mss,speed_ms,0,0.001)
    |   movel(pose_trans(ref_frame,p[0.031160, 0.018244, -0.000125, -0.013708, 3.141563, 0.000000]),accel_mss,speed_ms,0,0.001)
    |   movel(pose_trans(ref_frame,p[0.031066, 0.018324, -0.000125, -0.013708, 3.141563, -0.000000]),accel_mss,speed_ms,0,0.001)
    |   movel(pose_trans(ref_frame,p[0.030979, 0.018410, -0.000125, -0.013708, 3.141563, -0.000000]),accel_mss,speed_ms,0,0.001)
    |   movel(pose_trans(ref_frame,p[0.030850, 0.018552, -0.000125, -0.013708, 3.141563, -0.000000]),accel_mss,speed_ms,0,0.001)
    |   movel(pose_trans(ref_frame,p[0.030724, 0.018697, -0.000125, -0.013708, 3.141563, -0.000000]),accel_mss,speed_ms,0,0.001)
    |   movel(pose_trans(ref_frame,p[0.030360, 0.019190, -0.000125, -0.013708, 3.141563, -0.000000]),accel_mss,speed_ms,0,0.001)
    |   movel(pose_trans(ref_frame,p[0.030069, 0.019728, -0.000125, -0.013708, 3.141563, 0.000000]),accel_mss,speed_ms,0,0.001)
    |   movel(pose_trans(ref_frame,p[0.029840, 0.020324, -0.000125, -0.013708, 3.141563, -0.000000]),accel_mss,speed_ms,0,0.001)
    |   movel(pose_trans(ref_frame,p[0.029686, 0.020944, -0.000125, -0.013708, 3.141563, -0.000000]),accel_mss,speed_ms,0,0.001)
    |   movel(pose_trans(ref_frame,p[0.029559, 0.021816, -0.000125, -0.013708, 3.141563, 0.000000]),accel_mss,speed_ms,0,0.001)
    |   movel(pose_trans(ref_frame,p[0.029495, 0.022696, -0.000125, -0.013708, 3.141563, -0.000000]),accel_mss,speed_ms,0,0.001)
    |   movel(pose_trans(ref_frame,p[0.029456, 0.024175, -0.000125, -0.013708, 3.141563, -0.000000]),accel_mss,speed_ms,0,0.001)
    |   movel(pose_trans(ref_frame,p[0.029443, 0.025654, -0.000125, -0.013708, 3.141563, -0.000000]),accel_mss,speed_ms,0,0.001)
    |   movel(pose_trans(ref_frame,p[0.029440, 0.026652, -0.000125, -0.013708, 3.141563, -0.000000]),accel_mss,speed_ms,0,0.001)
    |   movel(pose_trans(ref_frame,p[0.029431, 0.027650, -0.000125, -0.013708, 3.141563, 0.000000]),accel_mss,speed_ms,0,0.001)
    |   movel(pose_trans(ref_frame,p[0.029417, 0.028201, -0.000125, -0.013708, 3.141563, 0.000000]),accel_mss,speed_ms,0,0.001)
    |   movel(pose_trans(ref_frame,p[0.029388, 0.028751, -0.000125, -0.013708, 3.141563, 0.000000]),accel_mss,speed_ms,0,0.001)
    |   movel(pose_trans(ref_frame,p[0.029354, 0.029121, -0.000125, -0.013708, 3.141563, 0.000000]),accel_mss,speed_ms,0,0.001)
    |   movel(pose_trans(ref_frame,p[0.029301, 0.029490, -0.000125, -0.013708, 3.141563, -0.000000]),accel_mss,speed_ms,0,0.001)
    |   movel(pose_trans(ref_frame,p[0.029235, 0.029801, -0.000125, -0.013708, 3.141563, -0.000000]),accel_mss,speed_ms,0,0.001)
    |   movel(pose_trans(ref_frame,p[0.029145, 0.030106, -0.000125, -0.013708, 3.141563, 0.000000]),accel_mss,speed_ms,0,0.001)
    |   movel(pose_trans(ref_frame,p[0.029054, 0.030362, -0.000125, -0.013708, 3.141563, 0.000000]),accel_mss,speed_ms,0,0.001)
    |   movel(pose_trans(ref_frame,p[0.028956, 0.030615, -0.000125, -0.013708, 3.141563, 0.000000]),accel_mss,speed_ms,0,0.001)
    |   movel(pose_trans(ref_frame,p[0.028884, 0.030773, -0.000125, -0.013708, 3.141563, -0.000000]),accel_mss,speed_ms,0,0.001)
    |   movel(pose_trans(ref_frame,p[0.028797, 0.030924, -0.000125, -0.013708, 3.141563, 0.000000]),accel_mss,speed_ms,0,0.001)
    |   movel(pose_trans(ref_frame,p[0.028698, 0.031061, -0.000125, -0.013708, 3.141563, 0.000000]),accel_mss,speed_ms,0,0.001)
    |   movel(pose_trans(ref_frame,p[0.028587, 0.031187, -0.000125, -0.013708, 3.141563, 0.000000]),accel_mss,speed_ms,0,0.001)
    |   movel(pose_trans(ref_frame,p[0.028411, 0.031360, -0.000125, -0.013708, 3.141563, 0.000000]),accel_mss,speed_ms,0,0.001)
    |   movel(pose_trans(ref_frame,p[0.028230, 0.031528, -0.000125, -0.013708, 3.141563, 0.000000]),accel_mss,speed_ms,0,0.001)
    |   movel(pose_trans(ref_frame,p[0.028052, 0.031682, -0.000125, -0.013708, 3.141563, -0.000000]),accel_mss,speed_ms,0,0.001)
    |   movel(pose_trans(ref_frame,p[0.027871, 0.031832, -0.000125, -0.013708, 3.141563, 0.000000]),accel_mss,speed_ms,0,0.001)
    |   movel(pose_trans(ref_frame,p[0.027754, 0.031915, -0.000125, -0.013708, 3.141563, -0.000000]),accel_mss,speed_ms,0,0.001)
    |   movel(pose_trans(ref_frame,p[0.027629, 0.031986, -0.000125, -0.013708, 3.141563, -0.000000]),accel_mss,speed_ms,0,0.001)
    |   movel(pose_trans(ref_frame,p[0.027517, 0.032033, -0.000125, -0.013708, 3.141563, 0.000000]),accel_mss,speed_ms,0,0.001)
    |   movel(pose_trans(ref_frame,p[0.027399, 0.032063, -0.000125, -0.013708, 3.141563, 0.000000]),accel_mss,speed_ms,0,0.001)
    |   movel(pose_trans(ref_frame,p[0.027250, 0.032083, -0.000125, -0.013708, 3.141563, -0.000000]),accel_mss,speed_ms,0,0.001)
    |   movel(pose_trans(ref_frame,p[0.027100, 0.032092, -0.000125, -0.013708, 3.141563, -0.000000]),accel_mss,speed_ms,0,0.001)
    |   movel(pose_trans(ref_frame,p[0.026855, 0.032083, -0.000125, -0.013708, 3.141563, 0.000000]),accel_mss,speed_ms,0,0.001)
    |   movel(pose_trans(ref_frame,p[0.026613, 0.032044, -0.000125, -0.013708, 3.141563, -0.000000]),accel_mss,speed_ms,0,0.001)
    |   movel(pose_trans(ref_frame,p[0.026391, 0.031978, -0.000125, -0.013708, 3.141563, -0.000000]),accel_mss,speed_ms,0,0.001)
    |   movel(pose_trans(ref_frame,p[0.026180, 0.031881, -0.000125, -0.013708, 3.141563, -0.000000]),accel_mss,speed_ms,0,0.001)
    |   movel(pose_trans(ref_frame,p[0.025993, 0.031760, -0.000125, -0.013708, 3.141563, -0.000000]),accel_mss,speed_ms,0,0.001)
    |   movel(pose_trans(ref_frame,p[0.025826, 0.031612, -0.000125, -0.013708, 3.141563, -0.000000]),accel_mss,speed_ms,0,0.001)
    |   movel(pose_trans(ref_frame,p[0.025684, 0.031443, -0.000125, -0.013708, 3.141563, -0.000000]),accel_mss,speed_ms,0,0.001)
    |   movel(pose_trans(ref_frame,p[0.025570, 0.031254, -0.000125, -0.013708, 3.141563, -0.000000]),accel_mss,speed_ms,0,0.001)
    |   movel(pose_trans(ref_frame,p[0.025505, 0.031104, -0.000125, -0.013708, 3.141563, -0.000000]),accel_mss,speed_ms,0,0.001)
    |   movel(pose_trans(ref_frame,p[0.025455, 0.030949, -0.000125, -0.013708, 3.141563, 0.000000]),accel_mss,speed_ms,0,0.001)
    |   movel(pose_trans(ref_frame,p[0.025450, 0.030849, -0.000125, -0.013708, 3.141563, -0.000000]),accel_mss,speed_ms,0,0.001)
    |   movel(pose_trans(ref_frame,p[0.025485, 0.030755, -0.000125, -0.013708, 3.141563, -0.000000]),accel_mss,speed_ms,0,0.001)
    |   movel(pose_trans(ref_frame,p[0.025559, 0.030672, -0.000125, -0.013708, 3.141563, -0.000000]),accel_mss,speed_ms,0,0.001)
    |   movel(pose_trans(ref_frame,p[0.025656, 0.030616, -0.000125, -0.013708, 3.141563, 0.000000]),accel_mss,speed_ms,0,0.001)
    |   movel(pose_trans(ref_frame,p[0.025852, 0.030550, -0.000125, -0.013708, 3.141563, -0.000000]),accel_mss,speed_ms,0,0.001)
    |   movel(pose_trans(ref_frame,p[0.026051, 0.030495, -0.000125, -0.013708, 3.141563, -0.000000]),accel_mss,speed_ms,0,0.001)
    |   movel(pose_trans(ref_frame,p[0.026360, 0.030386, -0.000125, -0.013708, 3.141563, -0.000000]),accel_mss,speed_ms,0,0.001)
    |   movel(pose_trans(ref_frame,p[0.026641, 0.030218, -0.000125, -0.013708, 3.141563, -0.000000]),accel_mss,speed_ms,0,0.001)
    |   movel(pose_trans(ref_frame,p[0.026895, 0.029990, -0.000125, -0.013708, 3.141563, 0.000000]),accel_mss,speed_ms,0,0.001)
    |   movel(pose_trans(ref_frame,p[0.027105, 0.029721, -0.000125, -0.013708, 3.141563, -0.000000]),accel_mss,speed_ms,0,0.001)
    |   movel(pose_trans(ref_frame,p[0.027267, 0.029412, -0.000125, -0.013708, 3.141563, -0.000000]),accel_mss,speed_ms,0,0.001)
    |   movel(pose_trans(ref_frame,p[0.027374, 0.029081, -0.000125, -0.013708, 3.141563, 0.000000]),accel_mss,speed_ms,0,0.001)
    |   movel(pose_trans(ref_frame,p[0.027420, 0.028738, -0.000125, -0.013708, 3.141563, -0.000000]),accel_mss,speed_ms,0,0.001)
    |   movel(pose_trans(ref_frame,p[0.027405, 0.028393, -0.000125, -0.013708, 3.141563, -0.000000]),accel_mss,speed_ms,0,0.001)
    |   movel(pose_trans(ref_frame,p[0.027339, 0.028097, -0.000125, -0.013708, 3.141563, -0.000000]),accel_mss,speed_ms,0,0.001)
    |   movel(pose_trans(ref_frame,p[0.027224, 0.027816, -0.000125, -0.013708, 3.141563, -0.000000]),accel_mss,speed_ms,0,0.001)
    |   movel(pose_trans(ref_frame,p[0.027053, 0.027526, -0.000125, -0.013708, 3.141563, 0.000000]),accel_mss,speed_ms,0,0.001)
    |   movel(pose_trans(ref_frame,p[0.026847, 0.027260, -0.000125, -0.013708, 3.141563, -0.000000]),accel_mss,speed_ms,0,0.001)
    |   movel(pose_trans(ref_frame,p[0.026606, 0.027017, -0.000125, -0.013708, 3.141563, -0.000000]),accel_mss,speed_ms,0,0.001)
    |   movel(pose_trans(ref_frame,p[0.026336, 0.026804, -0.000125, -0.013708, 3.141563, 0.000000]),accel_mss,speed_ms,0,0.001)
    |   movel(pose_trans(ref_frame,p[0.026059, 0.026642, -0.000125, -0.013708, 3.141563, 0.000000]),accel_mss,speed_ms,0,0.001)
    |   movel(pose_trans(ref_frame,p[0.025762, 0.026522, -0.000125, -0.013708, 3.141563, 0.000000]),accel_mss,speed_ms,0,0.001)
    |   movel(pose_trans(ref_frame,p[0.025463, 0.026444, -0.000125, -0.013708, 3.141563, -0.000000]),accel_mss,speed_ms,0,0.001)
    |   movel(pose_trans(ref_frame,p[0.025158, 0.026399, -0.000125, -0.013708, 3.141563, 0.000000]),accel_mss,speed_ms,0,0.001)
    |   movel(pose_trans(ref_frame,p[0.024895, 0.026398, -0.000125, -0.013708, 3.141563, -0.000000]),accel_mss,speed_ms,0,0.001)
    |   movel(pose_trans(ref_frame,p[0.024635, 0.026442, -0.000125, -0.013708, 3.141563, -0.000000]),accel_mss,speed_ms,0,0.001)
    |   movel(pose_trans(ref_frame,p[0.024393, 0.026529, -0.000125, -0.013708, 3.141563, 0.000000]),accel_mss,speed_ms,0,0.001)
    |   movel(pose_trans(ref_frame,p[0.024170, 0.026658, -0.000125, -0.013708, 3.141563, -0.000000]),accel_mss,speed_ms,0,0.001)
    |   movel(pose_trans(ref_frame,p[0.023940, 0.026841, -0.000125, -0.013708, 3.141563, -0.000000]),accel_mss,speed_ms,0,0.001)
    |   movel(pose_trans(ref_frame,p[0.023734, 0.027050, -0.000125, -0.013708, 3.141563, -0.000000]),accel_mss,speed_ms,0,0.001)
    |   movel(pose_trans(ref_frame,p[0.023331, 0.027704, -0.000125, -0.013708, 3.141563, 0.000000]),accel_mss,speed_ms,0,0.001)
    |   movel(pose_trans(ref_frame,p[0.023160, 0.028454, -0.000125, -0.013708, 3.141563, -0.000000]),accel_mss,speed_ms,0,0.001)
    |   movel(pose_trans(ref_frame,p[0.023209, 0.029312, -0.000125, -0.013708, 3.141563, -0.000000]),accel_mss,speed_ms,0,0.001)
    |   movel(pose_trans(ref_frame,p[0.023457, 0.030134, -0.000125, -0.013708, 3.141563, -0.000000]),accel_mss,speed_ms,0,0.001)
    |   movel(pose_trans(ref_frame,p[0.023973, 0.031085, -0.000125, -0.013708, 3.141563, -0.000000]),accel_mss,speed_ms,0,0.001)
    |   movel(pose_trans(ref_frame,p[0.024644, 0.031933, -0.000125, -0.013708, 3.141563, -0.000000]),accel_mss,speed_ms,0,0.001)
    |   movel(pose_trans(ref_frame,p[0.025585, 0.032837, -0.000125, -0.013708, 3.141563, -0.000000]),accel_mss,speed_ms,0,0.001)
    |   movel(pose_trans(ref_frame,p[0.026610, 0.033644, -0.000125, -0.013708, 3.141563, 0.000000]),accel_mss,speed_ms,0,0) # end trace
    |   speed_ms    = 1.000
    |   movel(pose_trans(ref_frame,p[0.026610, 0.033644, 0.005000, -0.013708, 3.141563, -0.000000]),accel_mss,speed_ms,0,0.001)
    |   movel(pose_trans(ref_frame,p[0.030968, 0.092934, 0.005000, -0.013708, 3.141563, 0.000000]),accel_mss,speed_ms,0,0) # end trace
    |   speed_ms    = 0.002
    |   movel(pose_trans(ref_frame,p[0.030968, 0.092934, -0.000125, -0.013708, 3.141563, -0.000000]),accel_mss,speed_ms,0,0) # end trace
    |   speed_ms    = 0.007
    |   movel(pose_trans(ref_frame,p[0.031315, 0.093192, -0.000125, -0.013708, 3.141563, 0.000000]),accel_mss,speed_ms,0,0.001)
    |   movel(pose_trans(ref_frame,p[0.031680, 0.093424, -0.000125, -0.013708, 3.141563, -0.000000]),accel_mss,speed_ms,0,0.001)
    |   movel(pose_trans(ref_frame,p[0.032051, 0.093627, -0.000125, -0.013708, 3.141563, -0.000000]),accel_mss,speed_ms,0,0.001)
    |   movel(pose_trans(ref_frame,p[0.032437, 0.093801, -0.000125, -0.013708, 3.141563, -0.000000]),accel_mss,speed_ms,0,0.001)
    |   movel(pose_trans(ref_frame,p[0.032880, 0.093967, -0.000125, -0.013708, 3.141563, 0.000000]),accel_mss,speed_ms,0,0.001)
    |   movel(pose_trans(ref_frame,p[0.033332, 0.094104, -0.000125, -0.013708, 3.141563, -0.000000]),accel_mss,speed_ms,0,0.001)
    |   movel(pose_trans(ref_frame,p[0.033898, 0.094246, -0.000125, -0.013708, 3.141563, 0.000000]),accel_mss,speed_ms,0,0.001)
    |   movel(pose_trans(ref_frame,p[0.034469, 0.094369, -0.000125, -0.013708, 3.141563, -0.000000]),accel_mss,speed_ms,0,0.001)
    |   movel(pose_trans(ref_frame,p[0.035555, 0.094585, -0.000125, -0.013708, 3.141563, -0.000000]),accel_mss,speed_ms,0,0.001)
    |   movel(pose_trans(ref_frame,p[0.035794, 0.095202, -0.000125, -0.013708, 3.141563, -0.000000]),accel_mss,speed_ms,0,0.001)
    |   movel(pose_trans(ref_frame,p[0.036053, 0.095865, -0.000125, -0.013708, 3.141563, -0.000000]),accel_mss,speed_ms,0,0.001)
    |   movel(pose_trans(ref_frame,p[0.036318, 0.096527, -0.000125, -0.013708, 3.141563, 0.000000]),accel_mss,speed_ms,0,0.001)
    |   movel(pose_trans(ref_frame,p[0.036444, 0.096812, -0.000125, -0.013708, 3.141563, -0.000000]),accel_mss,speed_ms,0,0.001)
    |   movel(pose_trans(ref_frame,p[0.036590, 0.097089, -0.000125, -0.013708, 3.141563, -0.000000]),accel_mss,speed_ms,0,0.001)
    |   movel(pose_trans(ref_frame,p[0.036731, 0.097308, -0.000125, -0.013708, 3.141563, -0.000000]),accel_mss,speed_ms,0,0.001)
    |   movel(pose_trans(ref_frame,p[0.036894, 0.097511, -0.000125, -0.013708, 3.141563, 0.000000]),accel_mss,speed_ms,0,0.001)
    |   movel(pose_trans(ref_frame,p[0.037161, 0.097801, -0.000125, -0.013708, 3.141563, -0.000000]),accel_mss,speed_ms,0,0.001)
    |   movel(pose_trans(ref_frame,p[0.037437, 0.098082, -0.000125, -0.013708, 3.141563, -0.000000]),accel_mss,speed_ms,0,0.001)
    |   movel(pose_trans(ref_frame,p[0.037935, 0.098534, -0.000125, -0.013708, 3.141563, 0.000000]),accel_mss,speed_ms,0,0.001)
    |   movel(pose_trans(ref_frame,p[0.038470, 0.098944, -0.000125, -0.013708, 3.141563, -0.000000]),accel_mss,speed_ms,0,0.001)
    |   movel(pose_trans(ref_frame,p[0.038984, 0.099263, -0.000125, -0.013708, 3.141563, -0.000000]),accel_mss,speed_ms,0,0.001)
    |   movel(pose_trans(ref_frame,p[0.039531, 0.099522, -0.000125, -0.013708, 3.141563, 0.000000]),accel_mss,speed_ms,0,0.001)
    |   movel(pose_trans(ref_frame,p[0.040098, 0.099716, -0.000125, -0.013708, 3.141563, -0.000000]),accel_mss,speed_ms,0,0.001)
    |   movel(pose_trans(ref_frame,p[0.040684, 0.099842, -0.000125, -0.013708, 3.141563, 0.000000]),accel_mss,speed_ms,0,0.001)
    |   movel(pose_trans(ref_frame,p[0.041336, 0.099915, -0.000125, -0.013708, 3.141563, -0.000000]),accel_mss,speed_ms,0,0.001)
    |   movel(pose_trans(ref_frame,p[0.041992, 0.099931, -0.000125, -0.013708, 3.141563, 0.000000]),accel_mss,speed_ms,0,0.001)
    |   movel(pose_trans(ref_frame,p[0.042354, 0.099911, -0.000125, -0.013708, 3.141563, -0.000000]),accel_mss,speed_ms,0,0.001)
    |   movel(pose_trans(ref_frame,p[0.042713, 0.099865, -0.000125, -0.013708, 3.141563, -0.000000]),accel_mss,speed_ms,0,0.001)
    |   movel(pose_trans(ref_frame,p[0.043135, 0.099787, -0.000125, -0.013708, 3.141563, 0.000000]),accel_mss,speed_ms,0,0.001)
    |   movel(pose_trans(ref_frame,p[0.043552, 0.099690, -0.000125, -0.013708, 3.141563, -0.000000]),accel_mss,speed_ms,0,0.001)
    |   movel(pose_trans(ref_frame,p[0.043965, 0.099576, -0.000125, -0.013708, 3.141563, -0.000000]),accel_mss,speed_ms,0,0.001)
    |   movel(pose_trans(ref_frame,p[0.044372, 0.099444, -0.000125, -0.013708, 3.141563, -0.000000]),accel_mss,speed_ms,0,0.001)
    |   movel(pose_trans(ref_frame,p[0.044711, 0.099312, -0.000125, -0.013708, 3.141563, 0.000000]),accel_mss,speed_ms,0,0.001)
    |   movel(pose_trans(ref_frame,p[0.045039, 0.099157, -0.000125, -0.013708, 3.141563, 0.000000]),accel_mss,speed_ms,0,0.001)
    |   movel(pose_trans(ref_frame,p[0.045781, 0.098710, -0.000125, -0.013708, 3.141563, 0.000000]),accel_mss,speed_ms,0,0.001)
    |   movel(pose_trans(ref_frame,p[0.046458, 0.098170, -0.000125, -0.013708, 3.141563, 0.000000]),accel_mss,speed_ms,0,0.001)
    |   movel(pose_trans(ref_frame,p[0.047110, 0.097509, -0.000125, -0.013708, 3.141563, -0.000000]),accel_mss,speed_ms,0,0.001)
    |   movel(pose_trans(ref_frame,p[0.047689, 0.096782, -0.000125, -0.013708, 3.141563, 0.000000]),accel_mss,speed_ms,0,0.001)
    |   movel(pose_trans(ref_frame,p[0.048168, 0.096027, -0.000125, -0.013708, 3.141563, 0.000000]),accel_mss,speed_ms,0,0.001)
    |   movel(pose_trans(ref_frame,p[0.048561, 0.095224, -0.000125, -0.013708, 3.141563, -0.000000]),accel_mss,speed_ms,0,0.001)
    |   movel(pose_trans(ref_frame,p[0.048799, 0.094493, -0.000125, -0.013708, 3.141563, -0.000000]),accel_mss,speed_ms,0,0.001)
    |   movel(pose_trans(ref_frame,p[0.048909, 0.093732, -0.000125, -0.013708, 3.141563, 0.000000]),accel_mss,speed_ms,0,0.001)
    |   movel(pose_trans(ref_frame,p[0.048937, 0.093413, -0.000125, -0.013708, 3.141563, -0.000000]),accel_mss,speed_ms,0,0.001)
    |   movel(pose_trans(ref_frame,p[0.048985, 0.093096, -0.000125, -0.013708, 3.141563, 0.000000]),accel_mss,speed_ms,0,0.001)
    |   movel(pose_trans(ref_frame,p[0.049045, 0.092903, -0.000125, -0.013708, 3.141563, 0.000000]),accel_mss,speed_ms,0,0.001)
    |   movel(pose_trans(ref_frame,p[0.049147, 0.092729, -0.000125, -0.013708, 3.141563, 0.000000]),accel_mss,speed_ms,0,0.001)
    |   movel(pose_trans(ref_frame,p[0.049304, 0.092554, -0.000125, -0.013708, 3.141563, -0.000000]),accel_mss,speed_ms,0,0.001)
    |   movel(pose_trans(ref_frame,p[0.049486, 0.092408, -0.000125, -0.013708, 3.141563, -0.000000]),accel_mss,speed_ms,0,0.001)
    |   movel(pose_trans(ref_frame,p[0.049899, 0.092134, -0.000125, -0.013708, 3.141563, 0.000000]),accel_mss,speed_ms,0,0.001)
    |   movel(pose_trans(ref_frame,p[0.050318, 0.091870, -0.000125, -0.013708, 3.141563, 0.000000]),accel_mss,speed_ms,0,0.001)
    |   movel(pose_trans(ref_frame,p[0.050561, 0.091716, -0.000125, -0.013708, 3.141563, -0.000000]),accel_mss,speed_ms,0,0.001)
    |   movel(pose_trans(ref_frame,p[0.050800, 0.091557, -0.000125, -0.013708, 3.141563, 0.000000]),accel_mss,speed_ms,0,0.001)
    |   movel(pose_trans(ref_frame,p[0.050985, 0.091424, -0.000125, -0.013708, 3.141563, -0.000000]),accel_mss,speed_ms,0,0.001)
    |   movel(pose_trans(ref_frame,p[0.051164, 0.091283, -0.000125, -0.013708, 3.141563, -0.000000]),accel_mss,speed_ms,0,0.001)
    |   movel(pose_trans(ref_frame,p[0.051320, 0.091145, -0.000125, -0.013708, 3.141563, 0.000000]),accel_mss,speed_ms,0,0.001)
    |   movel(pose_trans(ref_frame,p[0.051470, 0.090999, -0.000125, -0.013708, 3.141563, 0.000000]),accel_mss,speed_ms,0,0.001)
    |   movel(pose_trans(ref_frame,p[0.051624, 0.090833, -0.000125, -0.013708, 3.141563, 0.000000]),accel_mss,speed_ms,0,0.001)
    |   movel(pose_trans(ref_frame,p[0.051772, 0.090661, -0.000125, -0.013708, 3.141563, 0.000000]),accel_mss,speed_ms,0,0.001)
    |   movel(pose_trans(ref_frame,p[0.052351, 0.089856, -0.000125, -0.013708, 3.141563, -0.000000]),accel_mss,speed_ms,0,0.001)
    |   movel(pose_trans(ref_frame,p[0.052821, 0.088982, -0.000125, -0.013708, 3.141563, -0.000000]),accel_mss,speed_ms,0,0.001)
    |   movel(pose_trans(ref_frame,p[0.053129, 0.088128, -0.000125, -0.013708, 3.141563, 0.000000]),accel_mss,speed_ms,0,0.001)
    |   movel(pose_trans(ref_frame,p[0.053289, 0.087234, -0.000125, -0.013708, 3.141563, 0.000000]),accel_mss,speed_ms,0,0.001)
    |   movel(pose_trans(ref_frame,p[0.053299, 0.086309, -0.000125, -0.013708, 3.141563, -0.000000]),accel_mss,speed_ms,0,0.001)
    |   movel(pose_trans(ref_frame,p[0.053159, 0.085395, -0.000125, -0.013708, 3.141563, 0.000000]),accel_mss,speed_ms,0,0.001)
    |   movel(pose_trans(ref_frame,p[0.052860, 0.084401, -0.000125, -0.013708, 3.141563, 0.000000]),accel_mss,speed_ms,0,0.001)
    |   movel(pose_trans(ref_frame,p[0.052447, 0.083448, -0.000125, -0.013708, 3.141563, 0.000000]),accel_mss,speed_ms,0,0.001)
    |   movel(pose_trans(ref_frame,p[0.052114, 0.082828, -0.000125, -0.013708, 3.141563, 0.000000]),accel_mss,speed_ms,0,0.001)
    |   movel(pose_trans(ref_frame,p[0.051749, 0.082226, -0.000125, -0.013708, 3.141563, 0.000000]),accel_mss,speed_ms,0,0.001)
    |   movel(pose_trans(ref_frame,p[0.051337, 0.081616, -0.000125, -0.013708, 3.141563, -0.000000]),accel_mss,speed_ms,0,0.001)
    |   movel(pose_trans(ref_frame,p[0.050898, 0.081026, -0.000125, -0.013708, 3.141563, 0.000000]),accel_mss,speed_ms,0,0.001)
    |   movel(pose_trans(ref_frame,p[0.050316, 0.080305, -0.000125, -0.013708, 3.141563, 0.000000]),accel_mss,speed_ms,0,0.001)
    |   movel(pose_trans(ref_frame,p[0.049710, 0.079604, -0.000125, -0.013708, 3.141563, -0.000000]),accel_mss,speed_ms,0,0.001)
    |   movel(pose_trans(ref_frame,p[0.048815, 0.078613, -0.000125, -0.013708, 3.141563, -0.000000]),accel_mss,speed_ms,0,0.001)
    |   movel(pose_trans(ref_frame,p[0.047908, 0.077633, -0.000125, -0.013708, 3.141563, 0.000000]),accel_mss,speed_ms,0,0.001)
    |   movel(pose_trans(ref_frame,p[0.046950, 0.076598, -0.000125, -0.013708, 3.141563, 0.000000]),accel_mss,speed_ms,0,0.001)
    |   movel(pose_trans(ref_frame,p[0.046004, 0.075554, -0.000125, -0.013708, 3.141563, 0.000000]),accel_mss,speed_ms,0,0.001)
    |   movel(pose_trans(ref_frame,p[0.045372, 0.074828, -0.000125, -0.013708, 3.141563, 0.000000]),accel_mss,speed_ms,0,0.001)
    |   movel(pose_trans(ref_frame,p[0.044763, 0.074082, -0.000125, -0.013708, 3.141563, -0.000000]),accel_mss,speed_ms,0,0.001)
    |   movel(pose_trans(ref_frame,p[0.044257, 0.073416, -0.000125, -0.013708, 3.141563, -0.000000]),accel_mss,speed_ms,0,0.001)
    |   movel(pose_trans(ref_frame,p[0.043778, 0.072730, -0.000125, -0.013708, 3.141563, 0.000000]),accel_mss,speed_ms,0,0.001)
    |   movel(pose_trans(ref_frame,p[0.043253, 0.071925, -0.000125, -0.013708, 3.141563, -0.000000]),accel_mss,speed_ms,0,0.001)
    |   movel(pose_trans(ref_frame,p[0.042749, 0.071108, -0.000125, -0.013708, 3.141563, -0.000000]),accel_mss,speed_ms,0,0.001)
    |   movel(pose_trans(ref_frame,p[0.042025, 0.069852, -0.000125, -0.013708, 3.141563, -0.000000]),accel_mss,speed_ms,0,0.001)
    |   movel(pose_trans(ref_frame,p[0.041341, 0.068573, -0.000125, -0.013708, 3.141563, 0.000000]),accel_mss,speed_ms,0,0.001)
    |   movel(pose_trans(ref_frame,p[0.040742, 0.067355, -0.000125, -0.013708, 3.141563, 0.000000]),accel_mss,speed_ms,0,0.001)
    |   movel(pose_trans(ref_frame,p[0.040191, 0.066115, -0.000125, -0.013708, 3.141563, 0.000000]),accel_mss,speed_ms,0,0.001)
    |   movel(pose_trans(ref_frame,p[0.039735, 0.064965, -0.000125, -0.013708, 3.141563, -0.000000]),accel_mss,speed_ms,0,0.001)
    |   movel(pose_trans(ref_frame,p[0.039328, 0.063797, -0.000125, -0.013708, 3.141563, 0.000000]),accel_mss,speed_ms,0,0.001)
    |   movel(pose_trans(ref_frame,p[0.039023, 0.062751, -0.000125, -0.013708, 3.141563, 0.000000]),accel_mss,speed_ms,0,0.001)
    |   movel(pose_trans(ref_frame,p[0.038782, 0.061688, -0.000125, -0.013708, 3.141563, -0.000000]),accel_mss,speed_ms,0,0.001)
    |   movel(pose_trans(ref_frame,p[0.038642, 0.060684, -0.000125, -0.013708, 3.141563, -0.000000]),accel_mss,speed_ms,0,0.001)
    |   movel(pose_trans(ref_frame,p[0.038607, 0.059671, -0.000125, -0.013708, 3.141563, -0.000000]),accel_mss,speed_ms,0,0.001)
    |   movel(pose_trans(ref_frame,p[0.038679, 0.058647, -0.000125, -0.013708, 3.141563, -0.000000]),accel_mss,speed_ms,0,0.001)
    |   movel(pose_trans(ref_frame,p[0.038853, 0.057635, -0.000125, -0.013708, 3.141563, 0.000000]),accel_mss,speed_ms,0,0.001)
    |   movel(pose_trans(ref_frame,p[0.039132, 0.056635, -0.000125, -0.013708, 3.141563, -0.000000]),accel_mss,speed_ms,0,0.001)
    |   movel(pose_trans(ref_frame,p[0.039509, 0.055668, -0.000125, -0.013708, 3.141563, -0.000000]),accel_mss,speed_ms,0,0.001)
    |   movel(pose_trans(ref_frame,p[0.039983, 0.054736, -0.000125, -0.013708, 3.141563, 0.000000]),accel_mss,speed_ms,0,0.001)
    |   movel(pose_trans(ref_frame,p[0.040546, 0.053855, -0.000125, -0.013708, 3.141563, -0.000000]),accel_mss,speed_ms,0,0.001)
    |   movel(pose_trans(ref_frame,p[0.040987, 0.053317, -0.000125, -0.013708, 3.141563, 0.000000]),accel_mss,speed_ms,0,0.001)
    |   movel(pose_trans(ref_frame,p[0.041498, 0.052844, -0.000125, -0.013708, 3.141563, 0.000000]),accel_mss,speed_ms,0,0.001)
    |   movel(pose_trans(ref_frame,p[0.042059, 0.052455, -0.000125, -0.013708, 3.141563, 0.000000]),accel_mss,speed_ms,0,0.001)
    |   movel(pose_trans(ref_frame,p[0.042671, 0.052152, -0.000125, -0.013708, 3.141563, 0.000000]),accel_mss,speed_ms,0,0.001)
    |   movel(pose_trans(ref_frame,p[0.043281, 0.051957, -0.000125, -0.013708, 3.141563, 0.000000]),accel_mss,speed_ms,0,0.001)
    |   movel(pose_trans(ref_frame,p[0.043914, 0.051860, -0.000125, -0.013708, 3.141563, -0.000000]),accel_mss,speed_ms,0,0.001)
    |   movel(pose_trans(ref_frame,p[0.044501, 0.051875, -0.000125, -0.013708, 3.141563, -0.000000]),accel_mss,speed_ms,0,0.001)
    |   movel(pose_trans(ref_frame,p[0.045073, 0.052008, -0.000125, -0.013708, 3.141563, -0.000000]),accel_mss,speed_ms,0,0.001)
    |   movel(pose_trans(ref_frame,p[0.045276, 0.052083, -0.000125, -0.013708, 3.141563, 0.000000]),accel_mss,speed_ms,0,0.001)
    |   movel(pose_trans(ref_frame,p[0.045476, 0.052165, -0.000125, -0.013708, 3.141563, -0.000000]),accel_mss,speed_ms,0,0.001)
    |   movel(pose_trans(ref_frame,p[0.045614, 0.052234, -0.000125, -0.013708, 3.141563, -0.000000]),accel_mss,speed_ms,0,0.001)
    |   movel(pose_trans(ref_frame,p[0.045744, 0.052316, -0.000125, -0.013708, 3.141563, -0.000000]),accel_mss,speed_ms,0,0.001)
    |   movel(pose_trans(ref_frame,p[0.045872, 0.052417, -0.000125, -0.013708, 3.141563, -0.000000]),accel_mss,speed_ms,0,0.001)
    |   movel(pose_trans(ref_frame,p[0.045990, 0.052530, -0.000125, -0.013708, 3.141563, -0.000000]),accel_mss,speed_ms,0,0.001)
    |   movel(pose_trans(ref_frame,p[0.046164, 0.052716, -0.000125, -0.013708, 3.141563, -0.000000]),accel_mss,speed_ms,0,0.001)
    |   movel(pose_trans(ref_frame,p[0.046332, 0.052907, -0.000125, -0.013708, 3.141563, -0.000000]),accel_mss,speed_ms,0,0.001)
    |   movel(pose_trans(ref_frame,p[0.046882, 0.053666, -0.000125, -0.013708, 3.141563, 0.000000]),accel_mss,speed_ms,0,0.001)
    |   movel(pose_trans(ref_frame,p[0.047303, 0.054504, -0.000125, -0.013708, 3.141563, 0.000000]),accel_mss,speed_ms,0,0.001)
    |   movel(pose_trans(ref_frame,p[0.047696, 0.055607, -0.000125, -0.013708, 3.141563, -0.000000]),accel_mss,speed_ms,0,0.001)
    |   movel(pose_trans(ref_frame,p[0.047994, 0.056739, -0.000125, -0.013708, 3.141563, -0.000000]),accel_mss,speed_ms,0,0.001)
    |   movel(pose_trans(ref_frame,p[0.048289, 0.058300, -0.000125, -0.013708, 3.141563, -0.000000]),accel_mss,speed_ms,0,0.001)
    |   movel(pose_trans(ref_frame,p[0.048493, 0.059876, -0.000125, -0.013708, 3.141563, -0.000000]),accel_mss,speed_ms,0,0.001)
    |   movel(pose_trans(ref_frame,p[0.048696, 0.062146, -0.000125, -0.013708, 3.141563, 0.000000]),accel_mss,speed_ms,0,0.001)
    |   movel(pose_trans(ref_frame,p[0.048853, 0.064420, -0.000125, -0.013708, 3.141563, 0.000000]),accel_mss,speed_ms,0,0.001)
    |   movel(pose_trans(ref_frame,p[0.048882, 0.064887, -0.000125, -0.013708, 3.141563, -0.000000]),accel_mss,speed_ms,0,0.001)
    |   movel(pose_trans(ref_frame,p[0.048913, 0.065353, -0.000125, -0.013708, 3.141563, -0.000000]),accel_mss,speed_ms,0,0.001)
    |   movel(pose_trans(ref_frame,p[0.048947, 0.065818, -0.000125, -0.013708, 3.141563, -0.000000]),accel_mss,speed_ms,0,0.001)
    |   movel(pose_trans(ref_frame,p[0.048983, 0.066282, -0.000125, -0.013708, 3.141563, -0.000000]),accel_mss,speed_ms,0,0.001)
    |   movel(pose_trans(ref_frame,p[0.049016, 0.066687, -0.000125, -0.013708, 3.141563, -0.000000]),accel_mss,speed_ms,0,0.001)
    |   movel(pose_trans(ref_frame,p[0.049052, 0.067091, -0.000125, -0.013708, 3.141563, 0.000000]),accel_mss,speed_ms,0,0.001)
    |   movel(pose_trans(ref_frame,p[0.049077, 0.067333, -0.000125, -0.013708, 3.141563, 0.000000]),accel_mss,speed_ms,0,0.001)
    |   movel(pose_trans(ref_frame,p[0.049107, 0.067576, -0.000125, -0.013708, 3.141563, -0.000000]),accel_mss,speed_ms,0,0.001)
    |   movel(pose_trans(ref_frame,p[0.049138, 0.067813, -0.000125, -0.013708, 3.141563, -0.000000]),accel_mss,speed_ms,0,0.001)
    |   movel(pose_trans(ref_frame,p[0.049169, 0.068050, -0.000125, -0.013708, 3.141563, 0.000000]),accel_mss,speed_ms,0,0.001)
    |   movel(pose_trans(ref_frame,p[0.049218, 0.068430, -0.000125, -0.013708, 3.141563, -0.000000]),accel_mss,speed_ms,0,0.001)
    |   movel(pose_trans(ref_frame,p[0.049267, 0.068810, -0.000125, -0.013708, 3.141563, 0.000000]),accel_mss,speed_ms,0,0.001)
    |   movel(pose_trans(ref_frame,p[0.049321, 0.069241, -0.000125, -0.013708, 3.141563, 0.000000]),accel_mss,speed_ms,0,0.001)
    |   movel(pose_trans(ref_frame,p[0.049376, 0.069674, -0.000125, -0.013708, 3.141563, -0.000000]),accel_mss,speed_ms,0,0.001)
    |   movel(pose_trans(ref_frame,p[0.049429, 0.070102, -0.000125, -0.013708, 3.141563, 0.000000]),accel_mss,speed_ms,0,0.001)
    |   movel(pose_trans(ref_frame,p[0.049482, 0.070530, -0.000125, -0.013708, 3.141563, 0.000000]),accel_mss,speed_ms,0,0.001)
    |   movel(pose_trans(ref_frame,p[0.049606, 0.071498, -0.000125, -0.013708, 3.141563, 0.000000]),accel_mss,speed_ms,0,0.001)
    |   movel(pose_trans(ref_frame,p[0.049740, 0.072465, -0.000125, -0.013708, 3.141563, 0.000000]),accel_mss,speed_ms,0,0.001)
    |   movel(pose_trans(ref_frame,p[0.049882, 0.073423, -0.000125, -0.013708, 3.141563, 0.000000]),accel_mss,speed_ms,0,0.001)
    |   movel(pose_trans(ref_frame,p[0.050034, 0.074380, -0.000125, -0.013708, 3.141563, -0.000000]),accel_mss,speed_ms,0,0.001)
    |   movel(pose_trans(ref_frame,p[0.050174, 0.075208, -0.000125, -0.013708, 3.141563, 0.000000]),accel_mss,speed_ms,0,0.001)
    |   movel(pose_trans(ref_frame,p[0.050322, 0.076034, -0.000125, -0.013708, 3.141563, 0.000000]),accel_mss,speed_ms,0,0.001)
    |   movel(pose_trans(ref_frame,p[0.050421, 0.076513, -0.000125, -0.013708, 3.141563, -0.000000]),accel_mss,speed_ms,0,0.001)
    |   movel(pose_trans(ref_frame,p[0.050540, 0.076986, -0.000125, -0.013708, 3.141563, 0.000000]),accel_mss,speed_ms,0,0.001)
    |   movel(pose_trans(ref_frame,p[0.050859, 0.077888, -0.000125, -0.013708, 3.141563, -0.000000]),accel_mss,speed_ms,0,0.001)
    |   movel(pose_trans(ref_frame,p[0.051300, 0.078737, -0.000125, -0.013708, 3.141563, -0.000000]),accel_mss,speed_ms,0,0.001)
    |   movel(pose_trans(ref_frame,p[0.051869, 0.079543, -0.000125, -0.013708, 3.141563, 0.000000]),accel_mss,speed_ms,0,0.001)
    |   movel(pose_trans(ref_frame,p[0.052536, 0.080269, -0.000125, -0.013708, 3.141563, -0.000000]),accel_mss,speed_ms,0,0.001)
    |   movel(pose_trans(ref_frame,p[0.053333, 0.080947, -0.000125, -0.013708, 3.141563, 0.000000]),accel_mss,speed_ms,0,0.001)
    |   movel(pose_trans(ref_frame,p[0.054205, 0.081524, -0.000125, -0.013708, 3.141563, 0.000000]),accel_mss,speed_ms,0,0.001)
    |   movel(pose_trans(ref_frame,p[0.055203, 0.082040, -0.000125, -0.013708, 3.141563, 0.000000]),accel_mss,speed_ms,0,0.001)
    |   movel(pose_trans(ref_frame,p[0.056246, 0.082456, -0.000125, -0.013708, 3.141563, 0.000000]),accel_mss,speed_ms,0,0.001)
    |   movel(pose_trans(ref_frame,p[0.057206, 0.082740, -0.000125, -0.013708, 3.141563, -0.000000]),accel_mss,speed_ms,0,0.001)
    |   movel(pose_trans(ref_frame,p[0.058187, 0.082941, -0.000125, -0.013708, 3.141563, -0.000000]),accel_mss,speed_ms,0,0.001)
    |   movel(pose_trans(ref_frame,p[0.059198, 0.083061, -0.000125, -0.013708, 3.141563, -0.000000]),accel_mss,speed_ms,0,0.001)
    |   movel(pose_trans(ref_frame,p[0.060215, 0.083097, -0.000125, -0.013708, 3.141563, 0.000000]),accel_mss,speed_ms,0,0.001)
    |   movel(pose_trans(ref_frame,p[0.061192, 0.083050, -0.000125, -0.013708, 3.141563, -0.000000]),accel_mss,speed_ms,0,0.001)
    |   movel(pose_trans(ref_frame,p[0.062162, 0.082921, -0.000125, -0.013708, 3.141563, -0.000000]),accel_mss,speed_ms,0,0.001)
    |   movel(pose_trans(ref_frame,p[0.063026, 0.082717, -0.000125, -0.013708, 3.141563, -0.000000]),accel_mss,speed_ms,0,0.001)
    |   movel(pose_trans(ref_frame,p[0.063862, 0.082416, -0.000125, -0.013708, 3.141563, -0.000000]),accel_mss,speed_ms,0,0.001)
    |   movel(pose_trans(ref_frame,p[0.064062, 0.082325, -0.000125, -0.013708, 3.141563, -0.000000]),accel_mss,speed_ms,0,0.001)
    |   movel(pose_trans(ref_frame,p[0.064257, 0.082226, -0.000125, -0.013708, 3.141563, -0.000000]),accel_mss,speed_ms,0,0.001)
    |   movel(pose_trans(ref_frame,p[0.064422, 0.082131, -0.000125, -0.013708, 3.141563, 0.000000]),accel_mss,speed_ms,0,0.001)
    |   movel(pose_trans(ref_frame,p[0.064579, 0.082025, -0.000125, -0.013708, 3.141563, -0.000000]),accel_mss,speed_ms,0,0.001)
    |   movel(pose_trans(ref_frame,p[0.064743, 0.081899, -0.000125, -0.013708, 3.141563, -0.000000]),accel_mss,speed_ms,0,0.001)
    |   movel(pose_trans(ref_frame,p[0.064899, 0.081763, -0.000125, -0.013708, 3.141563, 0.000000]),accel_mss,speed_ms,0,0.001)
    |   movel(pose_trans(ref_frame,p[0.065100, 0.081573, -0.000125, -0.013708, 3.141563, 0.000000]),accel_mss,speed_ms,0,0.001)
    |   movel(pose_trans(ref_frame,p[0.065296, 0.081377, -0.000125, -0.013708, 3.141563, 0.000000]),accel_mss,speed_ms,0,0.001)
    |   movel(pose_trans(ref_frame,p[0.065576, 0.081070, -0.000125, -0.013708, 3.141563, 0.000000]),accel_mss,speed_ms,0,0.001)
    |   movel(pose_trans(ref_frame,p[0.065834, 0.080745, -0.000125, -0.013708, 3.141563, -0.000000]),accel_mss,speed_ms,0,0.001)
    |   movel(pose_trans(ref_frame,p[0.066061, 0.080409, -0.000125, -0.013708, 3.141563, -0.000000]),accel_mss,speed_ms,0,0.001)
    |   movel(pose_trans(ref_frame,p[0.066264, 0.080058, -0.000125, -0.013708, 3.141563, -0.000000]),accel_mss,speed_ms,0,0.001)
    |   movel(pose_trans(ref_frame,p[0.066464, 0.079647, -0.000125, -0.013708, 3.141563, 0.000000]),accel_mss,speed_ms,0,0.001)
    |   movel(pose_trans(ref_frame,p[0.066637, 0.079225, -0.000125, -0.013708, 3.141563, -0.000000]),accel_mss,speed_ms,0,0.001)
    |   movel(pose_trans(ref_frame,p[0.066829, 0.078684, -0.000125, -0.013708, 3.141563, -0.000000]),accel_mss,speed_ms,0,0.001)
    |   movel(pose_trans(ref_frame,p[0.067003, 0.078138, -0.000125, -0.013708, 3.141563, -0.000000]),accel_mss,speed_ms,0,0.001)
    |   movel(pose_trans(ref_frame,p[0.067260, 0.077286, -0.000125, -0.013708, 3.141563, 0.000000]),accel_mss,speed_ms,0,0.001)
    |   movel(pose_trans(ref_frame,p[0.067240, 0.077951, -0.000125, -0.013708, 3.141563, 0.000000]),accel_mss,speed_ms,0,0.001)
    |   movel(pose_trans(ref_frame,p[0.067233, 0.078140, -0.000125, -0.013708, 3.141563, -0.000000]),accel_mss,speed_ms,0,0.001)
    |   movel(pose_trans(ref_frame,p[0.067223, 0.078329, -0.000125, -0.013708, 3.141563, -0.000000]),accel_mss,speed_ms,0,0.001)
    |   movel(pose_trans(ref_frame,p[0.067201, 0.078670, -0.000125, -0.013708, 3.141563, 0.000000]),accel_mss,speed_ms,0,0.001)
    |   movel(pose_trans(ref_frame,p[0.067178, 0.079010, -0.000125, -0.013708, 3.141563, -0.000000]),accel_mss,speed_ms,0,0.001)
    |   movel(pose_trans(ref_frame,p[0.067149, 0.079408, -0.000125, -0.013708, 3.141563, -0.000000]),accel_mss,speed_ms,0,0.001)
    |   movel(pose_trans(ref_frame,p[0.067119, 0.079806, -0.000125, -0.013708, 3.141563, -0.000000]),accel_mss,speed_ms,0,0.001)
    |   movel(pose_trans(ref_frame,p[0.067087, 0.080214, -0.000125, -0.013708, 3.141563, -0.000000]),accel_mss,speed_ms,0,0.001)
    |   movel(pose_trans(ref_frame,p[0.067054, 0.080622, -0.000125, -0.013708, 3.141563, -0.000000]),accel_mss,speed_ms,0,0.001)
    |   movel(pose_trans(ref_frame,p[0.067006, 0.081263, -0.000125, -0.013708, 3.141563, 0.000000]),accel_mss,speed_ms,0,0.001)
    |   movel(pose_trans(ref_frame,p[0.066969, 0.081905, -0.000125, -0.013708, 3.141563, 0.000000]),accel_mss,speed_ms,0,0.001)
    |   movel(pose_trans(ref_frame,p[0.066969, 0.082238, -0.000125, -0.013708, 3.141563, -0.000000]),accel_mss,speed_ms,0,0.001)
    |   movel(pose_trans(ref_frame,p[0.067003, 0.082569, -0.000125, -0.013708, 3.141563, -0.000000]),accel_mss,speed_ms,0,0.001)
    |   movel(pose_trans(ref_frame,p[0.067055, 0.082722, -0.000125, -0.013708, 3.141563, -0.000000]),accel_mss,speed_ms,0,0.001)
    |   movel(pose_trans(ref_frame,p[0.067154, 0.082850, -0.000125, -0.013708, 3.141563, 0.000000]),accel_mss,speed_ms,0,0.001)
    |   movel(pose_trans(ref_frame,p[0.067274, 0.082908, -0.000125, -0.013708, 3.141563, -0.000000]),accel_mss,speed_ms,0,0.001)
    |   movel(pose_trans(ref_frame,p[0.067406, 0.082891, -0.000125, -0.013708, 3.141563, 0.000000]),accel_mss,speed_ms,0,0.001)
    |   movel(pose_trans(ref_frame,p[0.067541, 0.082804, -0.000125, -0.013708, 3.141563, -0.000000]),accel_mss,speed_ms,0,0.001)
    |   movel(pose_trans(ref_frame,p[0.067644, 0.082680, -0.000125, -0.013708, 3.141563, 0.000000]),accel_mss,speed_ms,0,0.001)
    |   movel(pose_trans(ref_frame,p[0.068118, 0.081892, -0.000125, -0.013708, 3.141563, -0.000000]),accel_mss,speed_ms,0,0.001)
    |   movel(pose_trans(ref_frame,p[0.068587, 0.081103, -0.000125, -0.013708, 3.141563, -0.000000]),accel_mss,speed_ms,0,0.001)
    |   movel(pose_trans(ref_frame,p[0.069075, 0.080265, -0.000125, -0.013708, 3.141563, 0.000000]),accel_mss,speed_ms,0,0.001)
    |   movel(pose_trans(ref_frame,p[0.069551, 0.079420, -0.000125, -0.013708, 3.141563, 0.000000]),accel_mss,speed_ms,0,0.001)
    |   movel(pose_trans(ref_frame,p[0.069991, 0.078613, -0.000125, -0.013708, 3.141563, -0.000000]),accel_mss,speed_ms,0,0.001)
    |   movel(pose_trans(ref_frame,p[0.070417, 0.077799, -0.000125, -0.013708, 3.141563, -0.000000]),accel_mss,speed_ms,0,0.001)
    |   movel(pose_trans(ref_frame,p[0.071339, 0.075937, -0.000125, -0.013708, 3.141563, -0.000000]),accel_mss,speed_ms,0,0.001)
    |   movel(pose_trans(ref_frame,p[0.072209, 0.074050, -0.000125, -0.013708, 3.141563, 0.000000]),accel_mss,speed_ms,0,0.001)
    |   movel(pose_trans(ref_frame,p[0.073173, 0.071823, -0.000125, -0.013708, 3.141563, 0.000000]),accel_mss,speed_ms,0,0.001)
    |   movel(pose_trans(ref_frame,p[0.074097, 0.069579, -0.000125, -0.013708, 3.141563, -0.000000]),accel_mss,speed_ms,0,0.001)
    |   movel(pose_trans(ref_frame,p[0.074941, 0.067421, -0.000125, -0.013708, 3.141563, 0.000000]),accel_mss,speed_ms,0,0.001)
    |   movel(pose_trans(ref_frame,p[0.075747, 0.065248, -0.000125, -0.013708, 3.141563, -0.000000]),accel_mss,speed_ms,0,0.001)
    |   movel(pose_trans(ref_frame,p[0.076281, 0.063655, -0.000125, -0.013708, 3.141563, -0.000000]),accel_mss,speed_ms,0,0.001)
    |   movel(pose_trans(ref_frame,p[0.076743, 0.062039, -0.000125, -0.013708, 3.141563, -0.000000]),accel_mss,speed_ms,0,0.001)
    |   movel(pose_trans(ref_frame,p[0.076955, 0.061230, -0.000125, -0.013708, 3.141563, 0.000000]),accel_mss,speed_ms,0,0.001)
    |   movel(pose_trans(ref_frame,p[0.078885, 0.059065, -0.000125, -0.013708, 3.141563, 0.000000]),accel_mss,speed_ms,0,0.001)
    |   movel(pose_trans(ref_frame,p[0.079446, 0.058444, -0.000125, -0.013708, 3.141563, -0.000000]),accel_mss,speed_ms,0,0.001)
    |   movel(pose_trans(ref_frame,p[0.080016, 0.057831, -0.000125, -0.013708, 3.141563, -0.000000]),accel_mss,speed_ms,0,0.001)
    |   movel(pose_trans(ref_frame,p[0.080693, 0.057119, -0.000125, -0.013708, 3.141563, -0.000000]),accel_mss,speed_ms,0,0.001)
    |   movel(pose_trans(ref_frame,p[0.081375, 0.056413, -0.000125, -0.013708, 3.141563, -0.000000]),accel_mss,speed_ms,0,0.001)
    |   movel(pose_trans(ref_frame,p[0.082204, 0.055569, -0.000125, -0.013708, 3.141563, -0.000000]),accel_mss,speed_ms,0,0.001)
    |   movel(pose_trans(ref_frame,p[0.083039, 0.054731, -0.000125, -0.013708, 3.141563, 0.000000]),accel_mss,speed_ms,0,0.001)
    |   movel(pose_trans(ref_frame,p[0.084077, 0.053700, -0.000125, -0.013708, 3.141563, 0.000000]),accel_mss,speed_ms,0,0.001)
    |   movel(pose_trans(ref_frame,p[0.085118, 0.052673, -0.000125, -0.013708, 3.141563, 0.000000]),accel_mss,speed_ms,0,0.001)
    |   movel(pose_trans(ref_frame,p[0.087346, 0.050467, -0.000125, -0.013708, 3.141563, -0.000000]),accel_mss,speed_ms,0,0.001)
    |   movel(pose_trans(ref_frame,p[0.089557, 0.048243, -0.000125, -0.013708, 3.141563, -0.000000]),accel_mss,speed_ms,0,0.001)
    |   movel(pose_trans(ref_frame,p[0.091137, 0.046610, -0.000125, -0.013708, 3.141563, -0.000000]),accel_mss,speed_ms,0,0.001)
    |   movel(pose_trans(ref_frame,p[0.092684, 0.044946, -0.000125, -0.013708, 3.141563, 0.000000]),accel_mss,speed_ms,0,0.001)
    |   movel(pose_trans(ref_frame,p[0.093888, 0.043588, -0.000125, -0.013708, 3.141563, -0.000000]),accel_mss,speed_ms,0,0.001)
    |   movel(pose_trans(ref_frame,p[0.095055, 0.042200, -0.000125, -0.013708, 3.141563, 0.000000]),accel_mss,speed_ms,0,0.001)
    |   movel(pose_trans(ref_frame,p[0.096077, 0.040904, -0.000125, -0.013708, 3.141563, 0.000000]),accel_mss,speed_ms,0,0.001)
    |   movel(pose_trans(ref_frame,p[0.097052, 0.039573, -0.000125, -0.013708, 3.141563, -0.000000]),accel_mss,speed_ms,0,0.001)
    |   movel(pose_trans(ref_frame,p[0.097732, 0.038559, -0.000125, -0.013708, 3.141563, -0.000000]),accel_mss,speed_ms,0,0.001)
    |   movel(pose_trans(ref_frame,p[0.098362, 0.037513, -0.000125, -0.013708, 3.141563, 0.000000]),accel_mss,speed_ms,0,0.001)
    |   movel(pose_trans(ref_frame,p[0.098835, 0.036597, -0.000125, -0.013708, 3.141563, -0.000000]),accel_mss,speed_ms,0,0.001)
    |   movel(pose_trans(ref_frame,p[0.099233, 0.035646, -0.000125, -0.013708, 3.141563, -0.000000]),accel_mss,speed_ms,0,0.001)
    |   movel(pose_trans(ref_frame,p[0.099514, 0.034768, -0.000125, -0.013708, 3.141563, -0.000000]),accel_mss,speed_ms,0,0.001)
    |   movel(pose_trans(ref_frame,p[0.099713, 0.033867, -0.000125, -0.013708, 3.141563, 0.000000]),accel_mss,speed_ms,0,0.001)
    |   movel(pose_trans(ref_frame,p[0.099821, 0.032974, -0.000125, -0.013708, 3.141563, 0.000000]),accel_mss,speed_ms,0,0.001)
    |   movel(pose_trans(ref_frame,p[0.099839, 0.032076, -0.000125, -0.013708, 3.141563, -0.000000]),accel_mss,speed_ms,0,0.001)
    |   movel(pose_trans(ref_frame,p[0.099730, 0.031042, -0.000125, -0.013708, 3.141563, -0.000000]),accel_mss,speed_ms,0,0.001)
    |   movel(pose_trans(ref_frame,p[0.099465, 0.030036, -0.000125, -0.013708, 3.141563, 0.000000]),accel_mss,speed_ms,0,0.001)
    |   movel(pose_trans(ref_frame,p[0.099058, 0.029127, -0.000125, -0.013708, 3.141563, -0.000000]),accel_mss,speed_ms,0,0.001)
    |   movel(pose_trans(ref_frame,p[0.098500, 0.028301, -0.000125, -0.013708, 3.141563, -0.000000]),accel_mss,speed_ms,0,0.001)
    |   movel(pose_trans(ref_frame,p[0.097794, 0.027564, -0.000125, -0.013708, 3.141563, -0.000000]),accel_mss,speed_ms,0,0.001)
    |   movel(pose_trans(ref_frame,p[0.096975, 0.026955, -0.000125, -0.013708, 3.141563, 0.000000]),accel_mss,speed_ms,0,0.001)
    |   movel(pose_trans(ref_frame,p[0.096001, 0.026437, -0.000125, -0.013708, 3.141563, -0.000000]),accel_mss,speed_ms,0,0.001)
    |   movel(pose_trans(ref_frame,p[0.094968, 0.026053, -0.000125, -0.013708, 3.141563, -0.000000]),accel_mss,speed_ms,0,0.001)
    |   movel(pose_trans(ref_frame,p[0.094408, 0.025907, -0.000125, -0.013708, 3.141563, -0.000000]),accel_mss,speed_ms,0,0.001)
    |   movel(pose_trans(ref_frame,p[0.093841, 0.025798, -0.000125, -0.013708, 3.141563, -0.000000]),accel_mss,speed_ms,0,0.001)
    |   movel(pose_trans(ref_frame,p[0.093171, 0.025706, -0.000125, -0.013708, 3.141563, 0.000000]),accel_mss,speed_ms,0,0.001)
    |   movel(pose_trans(ref_frame,p[0.092498, 0.025642, -0.000125, -0.013708, 3.141563, -0.000000]),accel_mss,speed_ms,0,0.001)
    |   movel(pose_trans(ref_frame,p[0.091870, 0.025605, -0.000125, -0.013708, 3.141563, -0.000000]),accel_mss,speed_ms,0,0.001)
    |   movel(pose_trans(ref_frame,p[0.091242, 0.025585, -0.000125, -0.013708, 3.141563, -0.000000]),accel_mss,speed_ms,0,0.001)
    |   movel(pose_trans(ref_frame,p[0.091023, 0.025626, -0.000125, -0.013708, 3.141563, -0.000000]),accel_mss,speed_ms,0,0.001)
    |   movel(pose_trans(ref_frame,p[0.090837, 0.025749, -0.000125, -0.013708, 3.141563, 0.000000]),accel_mss,speed_ms,0,0.001)
    |   movel(pose_trans(ref_frame,p[0.090776, 0.025835, -0.000125, -0.013708, 3.141563, -0.000000]),accel_mss,speed_ms,0,0.001)
    |   movel(pose_trans(ref_frame,p[0.090746, 0.025937, -0.000125, -0.013708, 3.141563, -0.000000]),accel_mss,speed_ms,0,0.001)
    |   movel(pose_trans(ref_frame,p[0.090742, 0.026077, -0.000125, -0.013708, 3.141563, 0.000000]),accel_mss,speed_ms,0,0.001)
    |   movel(pose_trans(ref_frame,p[0.090758, 0.026215, -0.000125, -0.013708, 3.141563, -0.000000]),accel_mss,speed_ms,0,0.001)
    |   movel(pose_trans(ref_frame,p[0.090807, 0.026407, -0.000125, -0.013708, 3.141563, -0.000000]),accel_mss,speed_ms,0,0.001)
    |   movel(pose_trans(ref_frame,p[0.090873, 0.026593, -0.000125, -0.013708, 3.141563, -0.000000]),accel_mss,speed_ms,0,0.001)
    |   movel(pose_trans(ref_frame,p[0.090985, 0.026849, -0.000125, -0.013708, 3.141563, -0.000000]),accel_mss,speed_ms,0,0.001)
    |   movel(pose_trans(ref_frame,p[0.091106, 0.027100, -0.000125, -0.013708, 3.141563, -0.000000]),accel_mss,speed_ms,0,0.001)
    |   movel(pose_trans(ref_frame,p[0.091297, 0.027522, -0.000125, -0.013708, 3.141563, -0.000000]),accel_mss,speed_ms,0,0.001)
    |   movel(pose_trans(ref_frame,p[0.091452, 0.027958, -0.000125, -0.013708, 3.141563, -0.000000]),accel_mss,speed_ms,0,0.001)
    |   movel(pose_trans(ref_frame,p[0.091513, 0.028279, -0.000125, -0.013708, 3.141563, -0.000000]),accel_mss,speed_ms,0,0.001)
    |   movel(pose_trans(ref_frame,p[0.091498, 0.028604, -0.000125, -0.013708, 3.141563, -0.000000]),accel_mss,speed_ms,0,0.001)
    |   movel(pose_trans(ref_frame,p[0.091408, 0.028951, -0.000125, -0.013708, 3.141563, -0.000000]),accel_mss,speed_ms,0,0.001)
    |   movel(pose_trans(ref_frame,p[0.091254, 0.029276, -0.000125, -0.013708, 3.141563, 0.000000]),accel_mss,speed_ms,0,0.001)
    |   movel(pose_trans(ref_frame,p[0.090938, 0.029779, -0.000125, -0.013708, 3.141563, 0.000000]),accel_mss,speed_ms,0,0.001)
    |   movel(pose_trans(ref_frame,p[0.090599, 0.030266, -0.000125, -0.013708, 3.141563, -0.000000]),accel_mss,speed_ms,0,0.001)
    |   movel(pose_trans(ref_frame,p[0.090259, 0.030698, -0.000125, -0.013708, 3.141563, 0.000000]),accel_mss,speed_ms,0,0.001)
    |   movel(pose_trans(ref_frame,p[0.089887, 0.031103, -0.000125, -0.013708, 3.141563, -0.000000]),accel_mss,speed_ms,0,0.001)
    |   movel(pose_trans(ref_frame,p[0.089089, 0.031901, -0.000125, -0.013708, 3.141563, -0.000000]),accel_mss,speed_ms,0,0.001)
    |   movel(pose_trans(ref_frame,p[0.088283, 0.032690, -0.000125, -0.013708, 3.141563, -0.000000]),accel_mss,speed_ms,0,0.001)
    |   movel(pose_trans(ref_frame,p[0.087421, 0.033514, -0.000125, -0.013708, 3.141563, -0.000000]),accel_mss,speed_ms,0,0.001)
    |   movel(pose_trans(ref_frame,p[0.086548, 0.034327, -0.000125, -0.013708, 3.141563, -0.000000]),accel_mss,speed_ms,0,0.001)
    |   movel(pose_trans(ref_frame,p[0.085830, 0.034970, -0.000125, -0.013708, 3.141563, 0.000000]),accel_mss,speed_ms,0,0.001)
    |   movel(pose_trans(ref_frame,p[0.085097, 0.035595, -0.000125, -0.013708, 3.141563, 0.000000]),accel_mss,speed_ms,0,0.001)
    |   movel(pose_trans(ref_frame,p[0.083811, 0.036667, -0.000125, -0.013708, 3.141563, -0.000000]),accel_mss,speed_ms,0,0.001)
    |   movel(pose_trans(ref_frame,p[0.082528, 0.037743, -0.000125, -0.013708, 3.141563, -0.000000]),accel_mss,speed_ms,0,0.001)
    |   movel(pose_trans(ref_frame,p[0.081839, 0.038332, -0.000125, -0.013708, 3.141563, -0.000000]),accel_mss,speed_ms,0,0.001)
    |   movel(pose_trans(ref_frame,p[0.081159, 0.038931, -0.000125, -0.013708, 3.141563, -0.000000]),accel_mss,speed_ms,0,0.001)
    |   movel(pose_trans(ref_frame,p[0.080666, 0.039385, -0.000125, -0.013708, 3.141563, -0.000000]),accel_mss,speed_ms,0,0.001)
    |   movel(pose_trans(ref_frame,p[0.080183, 0.039852, -0.000125, -0.013708, 3.141563, -0.000000]),accel_mss,speed_ms,0,0.001)
    |   movel(pose_trans(ref_frame,p[0.079687, 0.040357, -0.000125, -0.013708, 3.141563, -0.000000]),accel_mss,speed_ms,0,0.001)
    |   movel(pose_trans(ref_frame,p[0.079202, 0.040872, -0.000125, -0.013708, 3.141563, -0.000000]),accel_mss,speed_ms,0,0.001)
    |   movel(pose_trans(ref_frame,p[0.078933, 0.041162, -0.000125, -0.013708, 3.141563, -0.000000]),accel_mss,speed_ms,0,0.001)
    |   movel(pose_trans(ref_frame,p[0.078661, 0.041450, -0.000125, -0.013708, 3.141563, 0.000000]),accel_mss,speed_ms,0,0.001)
    |   movel(pose_trans(ref_frame,p[0.078450, 0.041668, -0.000125, -0.013708, 3.141563, -0.000000]),accel_mss,speed_ms,0,0.001)
    |   movel(pose_trans(ref_frame,p[0.078234, 0.041882, -0.000125, -0.013708, 3.141563, -0.000000]),accel_mss,speed_ms,0,0.001)
    |   movel(pose_trans(ref_frame,p[0.078070, 0.042040, -0.000125, -0.013708, 3.141563, 0.000000]),accel_mss,speed_ms,0,0.001)
    |   movel(pose_trans(ref_frame,p[0.077904, 0.042196, -0.000125, -0.013708, 3.141563, -0.000000]),accel_mss,speed_ms,0,0.001)
    |   movel(pose_trans(ref_frame,p[0.077891, 0.042202, -0.000125, -0.013708, 3.141563, -0.000000]),accel_mss,speed_ms,0,0.001)
    |   movel(pose_trans(ref_frame,p[0.077877, 0.042200, -0.000125, -0.013708, 3.141563, -0.000000]),accel_mss,speed_ms,0,0.001)
    |   movel(pose_trans(ref_frame,p[0.077866, 0.042191, -0.000125, -0.013708, 3.141563, 0.000000]),accel_mss,speed_ms,0,0.001)
    |   movel(pose_trans(ref_frame,p[0.077863, 0.042177, -0.000125, -0.013708, 3.141563, -0.000000]),accel_mss,speed_ms,0,0.001)
    |   movel(pose_trans(ref_frame,p[0.077867, 0.042123, -0.000125, -0.013708, 3.141563, -0.000000]),accel_mss,speed_ms,0,0.001)
    |   movel(pose_trans(ref_frame,p[0.077874, 0.042069, -0.000125, -0.013708, 3.141563, 0.000000]),accel_mss,speed_ms,0,0.001)
    |   movel(pose_trans(ref_frame,p[0.077898, 0.041904, -0.000125, -0.013708, 3.141563, 0.000000]),accel_mss,speed_ms,0,0.001)
    |   movel(pose_trans(ref_frame,p[0.077922, 0.041739, -0.000125, -0.013708, 3.141563, -0.000000]),accel_mss,speed_ms,0,0.001)
    |   movel(pose_trans(ref_frame,p[0.077951, 0.041544, -0.000125, -0.013708, 3.141563, -0.000000]),accel_mss,speed_ms,0,0.001)
    |   movel(pose_trans(ref_frame,p[0.077981, 0.041348, -0.000125, -0.013708, 3.141563, 0.000000]),accel_mss,speed_ms,0,0.001)
    |   movel(pose_trans(ref_frame,p[0.078016, 0.041131, -0.000125, -0.013708, 3.141563, -0.000000]),accel_mss,speed_ms,0,0.001)
    |   movel(pose_trans(ref_frame,p[0.078050, 0.040914, -0.000125, -0.013708, 3.141563, -0.000000]),accel_mss,speed_ms,0,0.001)
    |   movel(pose_trans(ref_frame,p[0.078398, 0.038489, -0.000125, -0.013708, 3.141563, -0.000000]),accel_mss,speed_ms,0,0.001)
    |   movel(pose_trans(ref_frame,p[0.078659, 0.036054, -0.000125, -0.013708, 3.141563, -0.000000]),accel_mss,speed_ms,0,0.001)
    |   movel(pose_trans(ref_frame,p[0.078750, 0.034207, -0.000125, -0.013708, 3.141563, -0.000000]),accel_mss,speed_ms,0,0.001)
    |   movel(pose_trans(ref_frame,p[0.078691, 0.032359, -0.000125, -0.013708, 3.141563, -0.000000]),accel_mss,speed_ms,0,0.001)
    |   movel(pose_trans(ref_frame,p[0.078506, 0.030891, -0.000125, -0.013708, 3.141563, -0.000000]),accel_mss,speed_ms,0,0.001)
    |   movel(pose_trans(ref_frame,p[0.078164, 0.029450, -0.000125, -0.013708, 3.141563, 0.000000]),accel_mss,speed_ms,0,0.001)
    |   movel(pose_trans(ref_frame,p[0.077696, 0.028208, -0.000125, -0.013708, 3.141563, 0.000000]),accel_mss,speed_ms,0,0.001)
    |   movel(pose_trans(ref_frame,p[0.077050, 0.027050, -0.000125, -0.013708, 3.141563, -0.000000]),accel_mss,speed_ms,0,0.001)
    |   movel(pose_trans(ref_frame,p[0.076799, 0.026687, -0.000125, -0.013708, 3.141563, 0.000000]),accel_mss,speed_ms,0,0.001)
    |   movel(pose_trans(ref_frame,p[0.076532, 0.026337, -0.000125, -0.013708, 3.141563, 0.000000]),accel_mss,speed_ms,0,0.001)
    |   movel(pose_trans(ref_frame,p[0.076275, 0.026035, -0.000125, -0.013708, 3.141563, -0.000000]),accel_mss,speed_ms,0,0.001)
    |   movel(pose_trans(ref_frame,p[0.076001, 0.025749, -0.000125, -0.013708, 3.141563, -0.000000]),accel_mss,speed_ms,0,0.001)
    |   movel(pose_trans(ref_frame,p[0.075700, 0.025472, -0.000125, -0.013708, 3.141563, -0.000000]),accel_mss,speed_ms,0,0.001)
    |   movel(pose_trans(ref_frame,p[0.075384, 0.025213, -0.000125, -0.013708, 3.141563, -0.000000]),accel_mss,speed_ms,0,0.001)
    |   movel(pose_trans(ref_frame,p[0.074999, 0.024928, -0.000125, -0.013708, 3.141563, 0.000000]),accel_mss,speed_ms,0,0.001)
    |   movel(pose_trans(ref_frame,p[0.074604, 0.024658, -0.000125, -0.013708, 3.141563, -0.000000]),accel_mss,speed_ms,0,0.001)
    |   movel(pose_trans(ref_frame,p[0.073734, 0.024146, -0.000125, -0.013708, 3.141563, -0.000000]),accel_mss,speed_ms,0,0.001)
    |   movel(pose_trans(ref_frame,p[0.072817, 0.023723, -0.000125, -0.013708, 3.141563, 0.000000]),accel_mss,speed_ms,0,0.001)
    |   movel(pose_trans(ref_frame,p[0.071855, 0.023390, -0.000125, -0.013708, 3.141563, -0.000000]),accel_mss,speed_ms,0,0.001)
    |   movel(pose_trans(ref_frame,p[0.070864, 0.023152, -0.000125, -0.013708, 3.141563, -0.000000]),accel_mss,speed_ms,0,0.001)
    |   movel(pose_trans(ref_frame,p[0.069817, 0.023003, -0.000125, -0.013708, 3.141563, 0.000000]),accel_mss,speed_ms,0,0.001)
    |   movel(pose_trans(ref_frame,p[0.068760, 0.022953, -0.000125, -0.013708, 3.141563, -0.000000]),accel_mss,speed_ms,0,0.001)
    |   movel(pose_trans(ref_frame,p[0.067639, 0.022996, -0.000125, -0.013708, 3.141563, -0.000000]),accel_mss,speed_ms,0,0.001)
    |   movel(pose_trans(ref_frame,p[0.066525, 0.023126, -0.000125, -0.013708, 3.141563, -0.000000]),accel_mss,speed_ms,0,0.001)
    |   movel(pose_trans(ref_frame,p[0.065452, 0.023347, -0.000125, -0.013708, 3.141563, -0.000000]),accel_mss,speed_ms,0,0.001)
    |   movel(pose_trans(ref_frame,p[0.064405, 0.023670, -0.000125, -0.013708, 3.141563, 0.000000]),accel_mss,speed_ms,0,0.001)
    |   movel(pose_trans(ref_frame,p[0.063330, 0.024108, -0.000125, -0.013708, 3.141563, -0.000000]),accel_mss,speed_ms,0,0.001)
    |   movel(pose_trans(ref_frame,p[0.062293, 0.024630, -0.000125, -0.013708, 3.141563, -0.000000]),accel_mss,speed_ms,0,0.001)
    |   movel(pose_trans(ref_frame,p[0.061342, 0.025211, -0.000125, -0.013708, 3.141563, -0.000000]),accel_mss,speed_ms,0,0.001)
    |   movel(pose_trans(ref_frame,p[0.060443, 0.025868, -0.000125, -0.013708, 3.141563, 0.000000]),accel_mss,speed_ms,0,0.001)
    |   movel(pose_trans(ref_frame,p[0.059735, 0.026510, -0.000125, -0.013708, 3.141563, -0.000000]),accel_mss,speed_ms,0,0.001)
    |   movel(pose_trans(ref_frame,p[0.059117, 0.027240, -0.000125, -0.013708, 3.141563, -0.000000]),accel_mss,speed_ms,0,0.001)
    |   movel(pose_trans(ref_frame,p[0.058740, 0.027818, -0.000125, -0.013708, 3.141563, 0.000000]),accel_mss,speed_ms,0,0.001)
    |   movel(pose_trans(ref_frame,p[0.058434, 0.028438, -0.000125, -0.013708, 3.141563, 0.000000]),accel_mss,speed_ms,0,0.001)
    |   movel(pose_trans(ref_frame,p[0.058223, 0.029057, -0.000125, -0.013708, 3.141563, -0.000000]),accel_mss,speed_ms,0,0.001)
    |   movel(pose_trans(ref_frame,p[0.058101, 0.029701, -0.000125, -0.013708, 3.141563, -0.000000]),accel_mss,speed_ms,0,0.001)
    |   movel(pose_trans(ref_frame,p[0.058087, 0.030217, -0.000125, -0.013708, 3.141563, -0.000000]),accel_mss,speed_ms,0,0.001)
    |   movel(pose_trans(ref_frame,p[0.058168, 0.030727, -0.000125, -0.013708, 3.141563, -0.000000]),accel_mss,speed_ms,0,0.001)
    |   movel(pose_trans(ref_frame,p[0.058340, 0.031051, -0.000125, -0.013708, 3.141563, -0.000000]),accel_mss,speed_ms,0,0.001)
    |   movel(pose_trans(ref_frame,p[0.058643, 0.031257, -0.000125, -0.013708, 3.141563, -0.000000]),accel_mss,speed_ms,0,0.001)
    |   movel(pose_trans(ref_frame,p[0.058764, 0.031289, -0.000125, -0.013708, 3.141563, -0.000000]),accel_mss,speed_ms,0,0.001)
    |   movel(pose_trans(ref_frame,p[0.058889, 0.031298, -0.000125, -0.013708, 3.141563, -0.000000]),accel_mss,speed_ms,0,0.001)
    |   movel(pose_trans(ref_frame,p[0.058988, 0.031278, -0.000125, -0.013708, 3.141563, 0.000000]),accel_mss,speed_ms,0,0.001)
    |   movel(pose_trans(ref_frame,p[0.059074, 0.031225, -0.000125, -0.013708, 3.141563, -0.000000]),accel_mss,speed_ms,0,0.001)
    |   movel(pose_trans(ref_frame,p[0.059153, 0.031133, -0.000125, -0.013708, 3.141563, -0.000000]),accel_mss,speed_ms,0,0.001)
    |   movel(pose_trans(ref_frame,p[0.059206, 0.031023, -0.000125, -0.013708, 3.141563, -0.000000]),accel_mss,speed_ms,0,0.001)
